METHOD PUBLIC CallBack : DINT
VAR_INPUT
  /// Response data
  RspData   : AxesGroupAcyclicAcrEntryRspBuffer;  
  /// Timestamp
  Timestamp : SystemTime;
END_VAR
// Create log entry
CreateLogMessage ( Timestamp   := Timestamp,
                   MessageType := MessageType.CMD,
                   Severity    := Severity.DEBUG,
                   MessageCode := 0,
                   MessageText := CONCAT('Callback reveiced in FB ', MyType));

ResponseData.Reset();
ResponseData.Payload    := RspData.Payload; 
ResponseData.PayloadLen := RspData.PayloadLen;
ParseResponsePayload( ResponseData :=  ResponseData , Timestamp := Timestamp);

// set flag for response received
_responseReceived := TRUE;
END_METHOD

METHOD PROTECTED CheckFunctionSupported : BOOL
VAR_IN_OUT
  /// Robot assignment of function
  AxesGroup : AxesGroup; 
END_VAR
Error   := TRUE;
ErrorID := RobotLibraryEvents.ERR_FUNCTION_NOT_SUPPORTED;

// Create log entry
CreateLogMessagePara1 ( Timestamp   := AxesGroup.InternalData.SystemTime,
                        MessageType := MessageType.CMD,
                        Severity    := Severity.DEBUG,
                        MessageCode := 0,
                        MessageText := 'Execution canceled, because function <{1}> is not supported by the robot controller',
                        Para1       :=  _myType);
END_METHOD

METHOD PROTECTED CheckParameterChanged : BOOL
VAR_IN_OUT
  /// Robot assignment of function
  AxesGroup    : AxesGroup; 
END_VAR
IF ( CheckParameterChanged )
THEN
  AxesGroup.Acyclic.ActiveCommandRegister.NotifyParameterChanged := _uniqueID;
END_IF
END_METHOD

METHOD PROTECTED CheckParameterValid : BOOL
VAR_IN_OUT
  /// Robot assignment of function
  AxesGroup : AxesGroup; 
END_VAR
CheckParameterValid := TRUE;
END_METHOD

METHOD INTERNAL CreateCommandPayload : RobotLibrarySendDataFB
VAR_IN_OUT
  /// Robot assignment of function
  AxesGroup    : AxesGroup; 
END_VAR
// Reset all variables
CreateCommandPayload.Reset();
// Add CmdType
CreateCommandPayload.AddUint(_cmdHeader.CmdTyp);
// Add Reserve_ExecMode
CreateCommandPayload.AddHalfBytes(  0               , _cmdHeader.ExecMode);
// Add ParSeq_Priority
CreateCommandPayload.AddHalfBytes( _cmdHeader.ParSeq, _cmdHeader.Priority);
END_METHOD

METHOD PROTECTED OnCall
VAR_IN_OUT
  /// Robot assignment of function
  AxesGroup         : AxesGroup; 
END_VAR
// map numeric value to enum, so that the corresponding message text is directly shown by the tooltip
ErrorIdEnum   := ErrorId;
WarningIdEnum := WarningId;
InfoIdEnum    := InfoId;

Error := ErrorID <> RobotLibraryConstants.OK;

ExternalLogger := AxesGroup.MessageLog.ExternalLogger;
LogLevel       := AxesGroup.MessageLog.LogLevel;

// building rising edges for error, warning, info number detected
_error_R  ( CLK := ErrorID   <> RobotLibraryConstants.OK );
_warning_R( CLK := WarningID <> RobotLibraryConstants.OK );
_info_R   ( CLK := InfoID    <> RobotLibraryConstants.OK );

IF ( _error_R.Q)
THEN
  // Create log entry
  CreateLogMessagePara2 ( Timestamp   := AxesGroup.InternalData.SystemTime,
                          MessageType := MessageType.CMD,
                          Severity    := Severity.DEBUG,
                          MessageCode := 0,
                          MessageText := 'Error with ID: 16#{1} in FB {2} received ',
                          Para1       := WORD_TO_STRING_HEX(ErrorID),
                          Para2       := MyType);                        
END_IF

IF ( _warning_R.Q)
THEN
  // Create log entry
  CreateLogMessagePara2 ( Timestamp   := AxesGroup.InternalData.SystemTime,
                          MessageType := MessageType.CMD,
                          Severity    := Severity.DEBUG,
                          MessageCode := 0,
                          MessageText := 'Warning with ID: 16#{1} in FB {2} received ',
                          Para1       := WORD_TO_STRING_HEX(WarningID),
                          Para2       := MyType);                        
END_IF

IF ( _info_R.Q)
THEN
  // Create log entry
  CreateLogMessagePara2 ( Timestamp   := AxesGroup.InternalData.SystemTime,
                          MessageType := MessageType.CMD,
                          Severity    := Severity.DEBUG,
                          MessageCode := 0,
                          MessageText := 'Info with ID: 16#{1} in FB {2} received ',
                          Para1       := WORD_TO_STRING_HEX(InfoID),
                          Para2       := MyType);                        
END_IF
END_METHOD

METHOD OnOnlineChange : DINT
VAR_IN_OUT
  /// Robot assignment of function
  AxesGroup : AxesGroup; 
END_VAR
// update pointer to command FB
AxesGroup.Acyclic.ActiveCommandRegister.OnOnlineChange( UniqueID := _uniqueID, pCommandFB := ADR(THIS^));
END_METHOD

METHOD INTERNAL ParseResponsePayload : DINT
VAR_INPUT
  /// Response data
  ResponseData : RobotLibraryRecvDataFB;
  /// Timestamp
  Timestamp    : SystemTime;  
END_VAR
// reset message IDs 
InfoID    := 0;
WarningID := 0;
ErrorID   := 0;

// get State
_rspHeader.State                := ResponseData.GetHalfeByte1(IncPayloadPtr := FALSE);
// get ParSeq
_rspHeader.ParSeq               := ResponseData.GetHalfeByte2(IncPayloadPtr := TRUE);
// get AlarmMessageSeverity
_rspHeader.AlarmMessageSeverity := ResponseData.GetSint();
// get AlarmMessageCode
_rspHeader.AlarmMessageCode     := ResponseData.GetUint();


// Update InfoID / WarningID / ErrorID
CASE _rspHeader.AlarmMessageSeverity OF

  // Informative message
  Severity.INFO        : InfoID    := _rspHeader.AlarmMessageCode;
  // Warning message
  Severity.WARNING     : WarningID := _rspHeader.AlarmMessageCode;
  // Error message
  Severity.ERROR       : ErrorID   := _rspHeader.AlarmMessageCode; 
  // Fataö error message
  Severity.FATAL_ERROR : ErrorID   := _rspHeader.AlarmMessageCode;

END_CASE

ParseResponsePayload := ResponseData.PayloadPtr;
END_METHOD

METHOD PROTECTED Reset : DINT
VAR_INPUT
END_VAR
_parameterUpdateInternal := FALSE;
_uniqueId := 0;
_stepCmd  := 0;
Error     := FALSE;
ErrorID   := 0;
WarningID := 0;
InfoID    := 0;  

Reset := RobotLibraryConstants.OK;
END_METHOD

END_FUNCTION_BLOCK

// Library/POUs/_internal/RobotLibraryRecvDataFB
{attribute 'pack_mode' := '1'} 
FUNCTION_BLOCK RobotLibraryRecvDataFB
// ------------------------------------------------------------------------- 
//  SRCI Robot Library                                                
// ------------------------------------------------------------------------- 
//                                                                           
//  Object:      RecvData                                       
//  Author:      Thorsten Brach                                                
//  Date:        2024-06-01
//
//  Description:                                              
//   
//                                                                           
//  Copyright: 
//    (C) 2024 Thorsten Brach. All rights reserved                                                                                                                                            
//             Licensed under the LGPL-3.0 license.
//                                                                           
//  Disclaimer:                                                                           
//    This project is provided without any guarantee and can be used for   
//    private and commercial purposes. Any use is at the user’s 
//    own risk and responsibility.
//
// -------------------------------------------------------------------------
VAR_INPUT
  /// Payload
  Payload    : ARRAY [0..RobotLibraryParameter.TELEGRAM_PAYLOAD_MAX] OF BYTE;
  /// Payload length
  PayloadLen : UDINT;
  /// Payload pointer
  PayloadPtr : DINT;
END_VAR

/// returns a ArmConfigParameter from the payload buffer from the current payload pointer address and increase the payload pointer afterwards
METHOD GetArmConfig : ArmConfigParameter
VAR
  /// temporary byte
 _tmpByte : BYTE;
END_VAR
// Table 5-17: Meaning of “Config” byte
// BIT 0 Shoulder TRUE : Shoulder is Back
//                FALSE: Shoulder is Front
// BIT 1 Elbow    TRUE : Elbow is Down
//                FALSE: Elbow is Up
// BIT 2 Wrist    TRUE : Wrist is Flip
//                FALSE: Wrist is Non-Flip
// BIT 3 Spare Not used
// BIT 4 Spare Not Used
// BIT 5 Spare Not Used
// BIT 6 Spare Not Used
// BIT 7 Spare Not Used
// get 1st Byte
_tmpByte := GetByte();

IF ( _tmpByte.0 ) 
THEN
  GetArmConfig.Shoulder := ArmConfigShoulder.BACK;
ELSE
  GetArmConfig.Shoulder := ArmConfigShoulder.FRONT;
END_IF

IF ( _tmpByte.1 ) 
THEN
  GetArmConfig.Elbow := ArmConfigElbow.DOWN;
ELSE
  GetArmConfig.Elbow := ArmConfigElbow.UP;
END_IF

IF ( _tmpByte.2 ) 
THEN
  GetArmConfig.Wrist := ArmConfigWrist.FLIP;
ELSE
  GetArmConfig.Wrist := ArmConfigWrist.NON_FLIP;
END_IF


// get 2nd byte to inc the PayloadPointer
_tmpByte := GetByte();
END_METHOD

/// returns a BOOL from the payload buffer from the current payload pointer address and increase the payload pointer afterwards
METHOD GetBool : BOOL
// copy data
GetBool := Payload[PayloadPtr].0;
// inc payload pointer 
PayloadPtr := PayloadPtr + SIZEOF(BYTE);
END_METHOD

/// returns a BYTE from the payload buffer from the current payload pointer address and increase the payload pointer afterwards
METHOD GetByte : BYTE
// copy data
GetByte := Payload[PayloadPtr];
// inc payload pointer 
PayloadPtr := PayloadPtr + SIZEOF(BYTE);
END_METHOD

/// returns a datablock from the payload buffer from the current payload pointer address and increase the payload pointer afterwards
METHOD GetDataBlock
VAR_INPUT
  /// Target
  pData    : POINTER TO BYTE;
  /// Size of data block
  Size     : UDINT;
  /// Target data type is string ? 
  IsString : BOOL;
END_VAR
IF ( pData <> RobotLibraryConstants.NULL_POINTER)
THEN
  IF ( IsString)
  THEN
    Size := Size -1;
  END_IF

  // copy data
  SysDepMemCpy(pDest := pData, pSrc := ADR(Payload[PayloadPtr]), DataLen := Size);
  
  // inc payload pointer 
  PayloadPtr := PayloadPtr + UDINT_TO_DINT(Size);
END_IF
END_METHOD

/// returns a DataInSync from the payload buffer from the current payload pointer address and increase the payload pointer afterwards
METHOD GetDataInSync : DataInSync
VAR
  /// temporary byte
 _tmpByte : BYTE;
END_VAR
// copy data
_tmpByte := Payload[PayloadPtr];

GetDataInSync.ToolsInSync             := _tmpByte.0;
GetDataInSync.FramesInSync            := _tmpByte.1;
GetDataInSync.LoadsInSync             := _tmpByte.2;
GetDataInSync.WorkAreasInSync         := _tmpByte.3;
GetDataInSync.SoftwareLimitsInSync    := _tmpByte.4;
GetDataInSync.DefaultDynamicsInSync   := _tmpByte.5;
GetDataInSync.ReferenceDynamicsInSync := _tmpByte.6;

// inc payload pointer   
PayloadPtr := PayloadPtr + SIZEOF(BYTE);
END_METHOD

/// returns a DWORD from the payload buffer from the current payload pointer address and increase the payload pointer afterwards
METHOD GetDword : DWORD
// copy data
SysDepMemCpy(pDest := ADR(GetDword), pSrc := ADR(Payload[PayloadPtr]), DataLen := SIZEOF(DWORD));
// inc payload pointer 
PayloadPtr := PayloadPtr + SIZEOF(DWORD);
END_METHOD

/// returns a FragmentAction from the payload buffer from the current payload pointer address and increase the payload pointer afterwards
METHOD GetFragmentAction : FragmentAction
VAR
  /// temporary byte
 _tmpByte : BYTE;
END_VAR
// copy data
_tmpByte := Payload[PayloadPtr];

GetFragmentAction.Complete := _tmpByte.0;
GetFragmentAction.Reset    := _tmpByte.1;
GetFragmentAction.Clear    := _tmpByte.2;
GetFragmentAction.BIT03    := _tmpByte.3;
GetFragmentAction.BIT04    := _tmpByte.4;
GetFragmentAction.BIT05    := _tmpByte.5;
GetFragmentAction.BIT06    := _tmpByte.6;
GetFragmentAction.BIT07    := _tmpByte.7;

// inc payload pointer   
PayloadPtr := PayloadPtr + SIZEOF(BYTE);
END_METHOD

/// returns the 1st halfe BYTE from the payload buffer from the current payload pointer address and increase the payload pointer afterwards
METHOD GetHalfeByte1 : BYTE
VAR_INPUT
  /// Increase payload pointer 
  IncPayloadPtr : BOOL;
END_VAR

VAR
  /// temporary byte
 _tmpByte : BYTE;
END_VAR
// copy data
_tmpByte := Payload[PayloadPtr];

GetHalfeByte1.0 := _tmpByte.0;
GetHalfeByte1.1 := _tmpByte.1;
GetHalfeByte1.2 := _tmpByte.2;
GetHalfeByte1.3 := _tmpByte.3;


IF (IncPayloadPtr)
THEN  
  // inc payload pointer
  PayloadPtr := PayloadPtr + SIZEOF(BYTE);
END_IF
END_METHOD

/// returns the 1st halfe BYTE from the payload buffer from the current payload pointer address and increase the payload pointer afterwards
METHOD GetHalfeByte2 : BYTE
VAR_INPUT
  /// Increase payload pointer 
  IncPayloadPtr : BOOL;
END_VAR

VAR
  /// temporary byte
 _tmpByte : BYTE;
END_VAR
// copy data
_tmpByte := Payload[PayloadPtr];

GetHalfeByte2.0 := _tmpByte.4;
GetHalfeByte2.1 := _tmpByte.5;
GetHalfeByte2.2 := _tmpByte.6;
GetHalfeByte2.3 := _tmpByte.7;

IF (IncPayloadPtr)
THEN  
  // inc payload pointer
  PayloadPtr := PayloadPtr + SIZEOF(BYTE);
END_IF
END_METHOD

/// returns a IEC_Date from the payload buffer from the current payload pointer address and increase the payload pointer afterwards
METHOD GetIecDate : IEC_Date
// copy data
SysDepMemCpy(pDest := ADR(GetIecDate), pSrc := ADR(Payload[PayloadPtr]), DataLen := SIZEOF(IEC_DATE));
// swap byte order
GetIecDate := SwapIecDate(GetIecDate);
// inc payload pointer   
PayloadPtr := PayloadPtr + SIZEOF(IEC_DATE);
END_METHOD

/// returns a IEC_TIME from the payload buffer from the current payload pointer address and increase the payload pointer afterwards
METHOD GetIecTime : IEC_TIME
// copy data
SysDepMemCpy(pDest := ADR(GetIecTime), pSrc := ADR(Payload[PayloadPtr]), DataLen := SIZEOF(IEC_TIME));
// swap byte order
GetIecTime := SwapIecTime(GetIecTime);
// inc payload pointer   
PayloadPtr := PayloadPtr + SIZEOF(IEC_TIME);
END_METHOD

/// returns a INT from the payload buffer from the current payload pointer address and increase the payload pointer afterwards
METHOD GetInt : INT
// copy data
SysDepMemCpy(pDest := ADR(GetInt), pSrc := ADR(Payload[PayloadPtr]), DataLen := SIZEOF(INT));
// swap byte order
GetInt := SwapInt(GetInt);
// inc payload pointer   
PayloadPtr := PayloadPtr + SIZEOF(INT);
END_METHOD

/// returns a REAL from the payload buffer from the current payload pointer address and increase the payload pointer afterwards
METHOD GetReal : REAL
// copy data
SysDepMemCpy(pDest := ADR(GetReal), pSrc := ADR(Payload[PayloadPtr]), DataLen := SIZEOF(REAL));
// swap byte order
GetReal := SwapReal(GetReal);
// inc payload pointer   
PayloadPtr := PayloadPtr + SIZEOF(Real);
END_METHOD

/// returns a SINT from the payload buffer from the current payload pointer address and increase the payload pointer afterwards
METHOD GetSint : SINT
// copy data
SysDepMemCpy(pDest := ADR(GetSint), pSrc := ADR(Payload[PayloadPtr]), DataLen := SIZEOF(SINT));
// inc payload pointer 
PayloadPtr := PayloadPtr + SIZEOF(SINT);
END_METHOD

/// returns a String from the payload buffer from the current payload pointer address and increase the payload pointer afterwards
METHOD GetString : STRING(255)
VAR_INPUT
  Size : DINT;
END_VAR
// copy data
SysDepMemCpy(pDest := ADR(GetString), pSrc := ADR(Payload[PayloadPtr]), DataLen := DINT_TO_UDINT(Size));

// inc payload pointer 
PayloadPtr := PayloadPtr + Size;
END_METHOD

/// returns a TrackingStatus from the payload buffer from the current payload pointer address and increase the payload pointer afterwards
METHOD GetTrackingStatus : TrackingStatus
VAR
  /// temporary byte
  tmpByte : BYTE;
END_VAR
// copy data
tmpByte := GetByte();

GetTrackingStatus.ConveyorTrackingEnabled   := tmpByte.0;  
GetTrackingStatus.WaitingForSynchronization := tmpByte.1;
GetTrackingStatus.Synchronizing             := tmpByte.2;
GetTrackingStatus.Synchronous               := tmpByte.3;
GetTrackingStatus.Desynchronizing           := tmpByte.4;
GetTrackingStatus.SyncOutZoneEntered        := tmpByte.5;
GetTrackingStatus.SyncOutZoneLeft           := tmpByte.6;
GetTrackingStatus.NotUsed                   := tmpByte.7;
END_METHOD

/// returns a TurnNumber from the payload buffer from the current payload pointer address and increase the payload pointer afterwards
METHOD GetTurnNumbers : TurnNumber
GetTurnNumbers.J1Turns := BYTE_TO_SINT(GetHalfeByte1(FALSE));
GetTurnNumbers.J2Turns := BYTE_TO_SINT(GetHalfeByte2(TRUE));

GetTurnNumbers.J3Turns := BYTE_TO_SINT(GetHalfeByte1(FALSE));
GetTurnNumbers.J4Turns := BYTE_TO_SINT(GetHalfeByte2(TRUE));

GetTurnNumbers.J5Turns := BYTE_TO_SINT(GetHalfeByte1(FALSE));
GetTurnNumbers.J6Turns := BYTE_TO_SINT(GetHalfeByte2(TRUE));

GetTurnNumbers.E1Turns := BYTE_TO_SINT(GetByte());
END_METHOD

/// returns a UDINT from the payload buffer from the current payload pointer address and increase the payload pointer afterwards
METHOD GetUdint : UDINT
// copy data
SysDepMemCpy(pDest := ADR(GetUdint), pSrc := ADR(Payload[PayloadPtr]), DataLen := SIZEOF(UDINT));
// swap byte order
GetUdint := SwapUdint(GetUdint);
// inc payload pointer   
PayloadPtr := PayloadPtr + SIZEOF(UDINT);
END_METHOD

/// returns a UINT from the payload buffer from the current payload pointer address and increase the payload pointer afterwards
METHOD GetUint : UINT
// copy data
SysDepMemCpy(pDest := ADR(GetUint), pSrc := ADR(Payload[PayloadPtr]), DataLen := SIZEOF(UINT));
// swap byte order
GetUint := SwapUint(GetUint);
// inc payload pointer   
PayloadPtr := PayloadPtr + SIZEOF(UINT);
END_METHOD

/// returns a USINT from the payload buffer from the current payload pointer address and increase the payload pointer afterwards
METHOD GetUsint : USINT
// copy data
SysDepMemCpy(pDest := ADR(GetUsint), pSrc := ADR(Payload[PayloadPtr]), DataLen := SIZEOF(USINT));
// inc payload pointer 
PayloadPtr := PayloadPtr + SIZEOF(USINT);
END_METHOD

/// returns a WORD from the payload buffer from the current payload pointer address and increase the payload pointer afterwards
METHOD GetWord : WORD
// copy data
SysDepMemCpy(pDest := ADR(GetWord), pSrc := ADR(Payload[PayloadPtr]), DataLen := SIZEOF(WORD));
// swap byte order
GetWord := SwapWord(GetWord);
// inc payload pointer   
PayloadPtr := PayloadPtr + SIZEOF(WORD);
END_METHOD

/// Resets the payload buffer, the payload pointer and the payload length
METHOD Reset
VAR_INPUT
END_VAR
SysDepMemSet(pDest := ADR(Payload), Value := 0 , DataLen := SIZEOF(Payload));
PayloadLen := 0;
PayloadPtr := 0;
END_METHOD

END_FUNCTION_BLOCK

// Library/POUs/_internal/AxesGroupMessageLogFB
FUNCTION_BLOCK AxesGroupMessageLogFB
// ------------------------------------------------------------------------- 
//  SRCI Robot Library                                                
// ------------------------------------------------------------------------- 
//                                                                           
//  Object:      AxesGroupMessageLogFB                                       
//  Author:      Thorsten Brach                                                
//  Date:        2025-01-05
//
//  Description:                                              
//   
//                                                                           
//  Copyright: 
//    (C) 2025 Thorsten Brach. All rights reserved                                                                                                                                            
//             Licensed under the LGPL-3.0 license.
//                                                                           
//  Disclaimer:                                                                           
//    This project is provided without any guarantee and can be used for   
//    private and commercial purposes. Any use is at the user’s 
//    own risk and responsibility.
//
// -------------------------------------------------------------------------
VAR_INPUT
  /// Logging level
  LogLevel         : LogLevel;
  /// Interface to an external logger
  ExternalLogger   : IMessageLogger;
END_VAR


VAR_OUTPUT
  /// Amount of system log entries
  SystemLogEntries : UINT := 0;
  /// Amount of message log entries
  MessagesEntries  : UINT := 0;
  /// System log
  SystemLogs       : ARRAY[0..RobotLibraryParameter.SYSTEM_LOG_MAX] OF STRING(255);
  /// Message Log
  Messages         : ARRAY[0..RobotLibraryParameter.MESSAGE_LOG_MAX] OF AlarmMessage;  
END_VAR

METHOD PUBLIC AddMessage
VAR_INPUT
  Message : ReadMessagesRecvData;
END_VAR

VAR
  /// internal index
 _idx            : DINT;
  /// internal index to delete
 _idxFound       : DINT;
  /// lowest Severity
 _lowestSeverity : Severity := Severity.FATAL_ERROR;
END_VAR
// Check entry must be added ? 
IF (( LogLevel  <= Message.Severity        ) AND
    ( LogLevel  >  LogLevelEnum.DEACTIVATE ))
THEN
  // Check message buffer is full ? 
  IF ( MessagesEntries >= RobotLibraryParameter.MESSAGE_LOG_MAX )
  THEN
    // find lowest Severity
    FOR _idx := 1 TO RobotLibraryParameter.MESSAGE_LOG_MAX
    DO
      // check entry has a lower severity ? 
     _lowestSeverity := MIN( Messages[_idx].Severity, _lowestSeverity );
		END_FOR

    // search for the oldes message with a lower Severity 
    FOR _idx := RobotLibraryParameter.MESSAGE_LOG_MAX TO 1 BY -1
    DO
      // message found ?
      IF (( Messages[_idx].Severity <  Message.Severity ) AND
          ( Messages[_idx].Severity <=  _lowestSeverity ))
      THEN
        // save index to delete 
       _idxFound := _idx;
        EXIT;
			END_IF
		END_FOR
    
    // check message must be deleted ? 
    IF ( _idxFound > 0 )
    THEN
      // shift all messages starting from the found index one position forwards
      FOR _idx := _idxFound TO RobotLibraryParameter.MESSAGE_LOG_MAX -1
      DO
        Messages[_idx] := Messages[_idx +1];
			END_FOR
		END_IF
  END_IF  


  // shift all messages one position backwards
  FOR _idx := RobotLibraryParameter.MESSAGE_LOG_MAX TO 1 BY -1
  DO
    Messages[_idx] := Messages[_idx-1]; 
  END_FOR

  // Add new message 
  Messages[0].Timestamp.SystemDate := IEC_DATE_TO_DATE(Message.Timestamp.IEC_DATE);           
  Messages[0].Timestamp.SystemTime := IEC_TIME_TO_TIME(Message.Timestamp.IEC_TIME);           
  Messages[0].MessageType          :=                  Message.MsgType;
  Messages[0].Severity             :=                  Message.Severity;
  Messages[0].MessageText          :=                  Message.Text;
  Messages[0].MessageCode          :=                  Message.ErrorCode;
  
  // inc message counter
  MessagesEntries := DINT_TO_UINT(LIMIT(0, MessagesEntries + 1, RobotLibraryParameter.MESSAGE_LOG_MAX));
END_IF
END_METHOD

METHOD PUBLIC AddSystemLog
VAR_INPUT
  SystemLog : STRING(255);
END_VAR

VAR
  /// internal index
 _idx : DINT;
END_VAR
FOR _idx := RobotLibraryParameter.SYSTEM_LOG_MAX TO 1 BY -1
DO
  SystemLogs[_idx] := SystemLogs[_idx-1]; 
END_FOR

SystemLogs[0] := SystemLog;           

// inc SystemLog counter
SystemLogEntries := DINT_TO_UINT(LIMIT(0, SystemLogEntries + 1, RobotLibraryParameter.SYSTEM_LOG_MAX));
END_METHOD

METHOD PUBLIC DeleteMessages
VAR_INPUT
END_VAR
// reset messages
SysDepMemSet(ADR(Messages), 0, SIZEOF(Messages));
// reset message counter
MessagesEntries := 0;
END_METHOD

METHOD DeleteSystemLogs
VAR_INPUT
END_VAR
// reset SystemLogs
SysDepMemSet(ADR(SystemLogs), 0, SIZEOF(SystemLogs));
// reset SystemLogs counter
SystemLogEntries := 0;
END_METHOD

END_FUNCTION_BLOCK

// Library/POUs/_internal/RobotLibraryBaseEnableFB
FUNCTION_BLOCK RobotLibraryBaseEnableFB EXTENDS RobotLibraryBaseFB
// ------------------------------------------------------------------------- 
//  SRCI Robot Library                                                
// ------------------------------------------------------------------------- 
//                                                                           
//  Object:      RobotLibraryBaseFB                                       
//  Author:      Thorsten Brach                                                
//  Date:        2024-08-11
//
//  Description:                                              
//   
//                                                                           
//  Copyright: 
//    (C) 2024 Thorsten Brach. All rights reserved                                                                                                                                            
//             Licensed under the LGPL-3.0 license.
//                                                                           
//  Disclaimer:                                                                           
//    This project is provided without any guarantee and can be used for   
//    private and commercial purposes. Any use is at the user’s 
//    own risk and responsibility.
//
// -------------------------------------------------------------------------
VAR_INPUT
  /// Set TRUE to activate / Set False to deactivate
  Enable            : BOOL;
END_VAR

VAR_OUTPUT
  /// FB is being processed
  Busy              : BOOL;
  /// Command is transferred and confirmed by the RC
//CommandBuffered   : BOOL;
  /// TRUE while function is active
  Enabled           : BOOL;
  /// Receiving of input parameter values has been acknowledged by RC
//ParameterAccepted : BOOL;
END_VAR

VAR
  /// step counter for finite state machine
 _fsmState          : FsmState;
  /// Rising edge for enable
 _enable_R          : R_TRIG;
  /// Falling edge for enable
 _enable_F          : F_TRIG;
END_VAR

SUPER^(AxesGroup := AxesGroup);

METHOD INTERNAL FSM : DINT
VAR_IN_OUT
  /// Robot assignment of function
  AxesGroup : AxesGroup; 
END_VAR
VAR
  /// internal return value
 _retVal : DINT;
END_VAR
CASE _fsmState 
OF

  FsmState.READY :
  
    // Await start
    IF (( NOT Busy       ) AND 
        ( NOT Error      ) AND 
        (    _enable_R.Q ))
    THEN
      // inc fsm step
     _fsmState := FsmState.START;
    END_IF
      
  FsmState.START :
   
   _retVal := OnExecStart(AxesGroup := AxesGroup);
    
    IF ( _retVal = RobotLibraryConstants.OK )
    THEN
     _fsmState := FsmState.RUNNING;
    ELSE
      // Cancel
      IF ((      Busy       ) AND
          (  NOT Error      ) AND
          (     _enable_F.Q ))
      THEN
       _fsmState := FsmState.CANCEL;
        RETURN;
      END_IF
    
      // check error 
      IF (_retVal < RobotLibraryConstants.OK)
      THEN
       _fsmState := FsmState.ERROR;
        RETURN;
      END_IF
    END_IF

   FsmState.RUNNING :

      _retVal := OnExecRun(AxesGroup := AxesGroup);
    
       IF (_retVal = RobotLibraryConstants.OK )
       THEN
        _fsmState := FsmState.DONE;
       ELSE
         // Cancel
         IF ((      Busy       ) AND
             (  NOT Error      ) AND
             (     _enable_F.Q ))
         THEN
          _fsmState := FsmState.CANCEL;
           RETURN;
         END_IF
         
         // error 
         IF (_retVal < RobotLibraryConstants.OK)
         THEN
          _fsmState := 99;
           RETURN;
         END_IF         
       END_IF

  FsmState.DONE :
  
   _fsmState := FsmState.READY;

  FsmState.CANCEL :

   _retVal := OnExecCancel(AxesGroup := AxesGroup);
    
    IF (_retVal = RobotLibraryConstants.OK )
    THEN
      _fsmState := FsmState.READY;
    END_IF
    
  FsmState.ERROR :
  
    IF (NOT Enable)
    THEN
     _fsmState := FsmState.ERROR_CLEAR;
    END_IF

  FsmState.ERROR_CLEAR :

   _retVal := OnExecErrorClear(AxesGroup := AxesGroup);
    
    IF (_retVal = RobotLibraryConstants.OK )
    THEN
      _fsmState := FsmState.READY;
    END_IF
       
ELSE
  ;
END_CASE
END_METHOD

METHOD PROTECTED OnCall
VAR_IN_OUT
  /// Robot assignment of function
  AxesGroup         : AxesGroup; 
END_VAR
SUPER^.OnCall(AxesGroup := AxesGroup);

// building rising and falling edges
_enable_R( CLK := Enable);
_enable_F( CLK := Enable);

// call state machine
FSM(AxesGroup := AxesGroup);


// Abort execution 
IF (Busy) AND ( _enable_F.Q) 
THEN
  // try to remove cmd
  AxesGroup.Acyclic.ActiveCommandRegister.RemoveCmd(_uniqueID);
END_IF
END_METHOD

METHOD Protected OnExecCancel : DINT
VAR_IN_OUT
  /// Robot assignment of function
  AxesGroup : AxesGroup; 
END_VAR
OnExecCancel := Reset();


// Create log entry
CreateLogMessagePara1 ( Timestamp   := AxesGroup.InternalData.SystemTime,
                        MessageType := MessageType.CMD,
                        Severity    := Severity.DEBUG,
                        MessageCode := 0,
                        MessageText := 'Execution of FB {1} cancled ',
                        Para1       := MyType);
END_METHOD

METHOD PROTECTED OnExecErrorClear : DINT
VAR_IN_OUT
  /// Robot assignment of function
  AxesGroup : AxesGroup; 
END_VAR
Reset();
END_METHOD

METHOD PROTECTED OnExecRun : DINT
VAR_IN_OUT
  /// Robot assignment of function
  AxesGroup : AxesGroup; 
END_VAR
END_METHOD

METHOD PROTECTED OnExecStart : DINT
VAR_IN_OUT
  /// Robot assignment of function
  AxesGroup : AxesGroup; 
END_VAR
END_METHOD

METHOD PROTECTED Reset : DINT
VAR_INPUT
END_VAR
Reset := SUPER^.Reset();

Busy    := FALSE;
Enabled := FALSE;
END_METHOD

END_FUNCTION_BLOCK

// Library/POUs/_internal/RobotLibraryBaseExecuteFB
FUNCTION_BLOCK RobotLibraryBaseExecuteFB EXTENDS RobotLibraryBaseFB
// ------------------------------------------------------------------------- 
//  SRCI Robot Library                                                
// ------------------------------------------------------------------------- 
//                                                                           
//  Object:      RobotLibraryBaseFB                                       
//  Author:      Thorsten Brach                                                
//  Date:        2024-08-11
//
//  Description:                                              
//   
//                                                                           
//  Copyright: 
//    (C) 2024 Thorsten Brach. All rights reserved                                                                                                                                            
//             Licensed under the LGPL-3.0 license.
//                                                                           
//  Disclaimer:                                                                           
//    This project is provided without any guarantee and can be used for   
//    private and commercial purposes. Any use is at the user’s 
//    own risk and responsibility.
//
// -------------------------------------------------------------------------
VAR_INPUT
  /// Start of the command at the rising edge
  Execute         : BOOL;
END_VAR
VAR_OUTPUT
  /// The command has been completed successfully
  Done            : BOOL;
  /// FB is being processed
  Busy            : BOOL;
  /// Command is transferred and confirmed by the RC
//  CommandBuffered : BOOL;  
END_VAR


VAR
  /// step counter for finite state machine
 _fsmState        : FsmState;
  /// Rising edge for execute
 _execute_R       : R_TRIG;
  /// Falling edge for execute
 _execute_F       : F_TRIG;
END_VAR

SUPER^(AxesGroup := AxesGroup);

METHOD internal FSM : DINT
VAR_IN_OUT
  /// Robot assignment of function
  AxesGroup : AxesGroup; 
END_VAR
VAR
  /// internal return value
 _retVal : DINT;
END_VAR
CASE _fsmState 
OF

  FsmState.READY :
  
    // Await start
    IF (( NOT Busy        ) AND 
        ( NOT Error       ) AND 
        (    _execute_R.Q ))
    THEN
      // inc fsm step
     _fsmState := FsmState.START;
    END_IF
      
  FsmState.START :
   
   _retVal := OnExecStart(AxesGroup := AxesGroup);
    
    IF ( _retVal = RobotLibraryConstants.OK )
    THEN
     _fsmState := FsmState.RUNNING;
    ELSE
      // Cancel
      IF ((      Busy        ) AND
          (  NOT Error       ) AND
          (     _execute_F.Q ))
      THEN
       _fsmState := FsmState.CANCEL;
        RETURN;
      END_IF
    
      // check error 
      IF (_retVal < RobotLibraryConstants.OK)
      THEN
       _fsmState := FsmState.ERROR;
        RETURN;
      END_IF
    END_IF

   FsmState.RUNNING :

      _retVal := OnExecRun(AxesGroup := AxesGroup);
    
       IF (_retVal = RobotLibraryConstants.OK )
       THEN
        _fsmState := FsmState.DONE;
       ELSE
         // Cancel
         IF ((      Busy        ) AND
             (  NOT Error       ) AND
             (     _execute_F.Q ))
         THEN
          _fsmState := FsmState.CANCEL;
           RETURN;
         END_IF
         
         // error 
         IF (_retVal < RobotLibraryConstants.OK)
         THEN
          _fsmState := 99;
           RETURN;
         END_IF         
       END_IF

  FsmState.DONE :
  
   _fsmState := FsmState.READY;

  FsmState.CANCEL :

   _retVal := OnExecCancel(AxesGroup := AxesGroup);
    
    IF (_retVal = RobotLibraryConstants.OK )
    THEN
      _fsmState := FsmState.READY;
    END_IF
    
  FsmState.ERROR :
  
    IF (NOT Execute)
    THEN
     _fsmState := FsmState.ERROR_CLEAR;
    END_IF

  FsmState.ERROR_CLEAR :

   _retVal := OnExecErrorClear(AxesGroup := AxesGroup);
    
    IF (_retVal = RobotLibraryConstants.OK )
    THEN
      _fsmState := FsmState.READY;
    END_IF
       
ELSE
  ;
END_CASE
END_METHOD

// Base implementation must be called ! 
METHOD PROTECTED OnCall
VAR_IN_OUT
  /// Robot assignment of function
  AxesGroup         : AxesGroup; 
END_VAR
SUPER^.OnCall(AxesGroup := AxesGroup);

// building rising and falling edges
_execute_R( CLK := Execute);
_execute_F( CLK := EXecute);

// call state machine
FSM(AxesGroup := AxesGroup);

// Abort execution 
IF (Busy) AND (_execute_F.Q) 
THEN
  // try to remove cmd
  AxesGroup.Acyclic.ActiveCommandRegister.RemoveCmd(_uniqueID);
END_IF
END_METHOD

METHOD PROTECTED OnExecCancel : DINT
VAR_IN_OUT
  /// Robot assignment of function
  AxesGroup : AxesGroup; 
END_VAR
OnExecCancel := Reset();


// Create log entry
CreateLogMessagePara1 ( Timestamp   := AxesGroup.InternalData.SystemTime,
                        MessageType := MessageType.CMD,
                        Severity    := Severity.DEBUG,
                        MessageCode := 0,
                        MessageText := 'Execution of FB {1} cancled ',
                        Para1       := MyType);
END_METHOD

METHOD PROTECTED OnExecErrorClear : DINT
VAR_IN_OUT
  /// Robot assignment of function
  AxesGroup : AxesGroup; 
END_VAR
Reset();
END_METHOD

METHOD PROTECTED OnExecRun : DINT
VAR_IN_OUT
  /// Robot assignment of function
  AxesGroup : AxesGroup; 
END_VAR
END_METHOD

METHOD PROTECTED OnExecStart : DINT
VAR_IN_OUT
  /// Robot assignment of function
  AxesGroup : AxesGroup; 
END_VAR
END_METHOD

METHOD PROTECTED Reset : DINT
VAR_INPUT
END_VAR
Reset := SUPER^.Reset();

Done := FALSE;
Busy := FALSE;
END_METHOD

END_FUNCTION_BLOCK

// Library/POUs/Additional/MC_AbortMeasuringInput/MC_AbortMeasuringInputFB
/// Abort triggering of Position, measuring input
FUNCTION_BLOCK MC_AbortMeasuringInputFB EXTENDS RobotLibraryBaseExecuteFB
// ------------------------------------------------------------------------- 
//  SRCI Robot Library                                                
// ------------------------------------------------------------------------- 
//                                                                           
//  Object:      AbortMeasuringInputFB                                       
//  Author:      Thorsten Brach                                                
//  Date:        2024-06-01
//
//  Description:                                              
//   
//                                                                           
//  Copyright: 
//    (C) 2024 Thorsten Brach. All rights reserved                                                                                                                                            
//             Licensed under the LGPL-3.0 license.
//                                                                           
//  Disclaimer:                                                                           
//    This project is provided without any guarantee and can be used for   
//    private and commercial purposes. Any use is at the user’s 
//    own risk and responsibility.
//
// -------------------------------------------------------------------------
VAR_INPUT
  /// Command parameter 
  ParCmd          : AbortMeasuringInputParCmd;      
END_VAR
VAR_OUTPUT
  /// Command is transferred and confirmed by the RC
  CommandBuffered : BOOL;  
  /// Command output 
  OutCmd          : AbortMeasuringInputOutCmd;          
END_VAR
VAR
  /// internal copy of command parameter 
 _parCmd          : AbortMeasuringInputParCmd;
  /// command data to send
 _command         : AbortMeasuringInputSendData;
  /// response data received
 _response        : AbortMeasuringInputRecvData;      
END_VAR

SUPER^(AxesGroup := AxesGroup);

METHOD PROTECTED CheckFunctionSupported : BOOL
VAR_IN_OUT
  /// Robot assignment of function
  AxesGroup : AxesGroup; 
END_VAR
CheckFunctionSupported := AxesGroup.InternalData.RCSupportedFunctions.AbortMeasuringInput;

IF ( NOT CheckFunctionSupported )
THEN
  // call base implementation for set error and create log entry
  SUPER^.CheckFunctionSupported(AxesGroup := AxesGroup);
END_IF
END_METHOD

METHOD PROTECTED CheckParameterChanged : BOOL
VAR_IN_OUT
  /// Robot assignment of function
  AxesGroup    : AxesGroup; 
END_VAR
// Check ParCmd Size is > 0, because MemCmp does not work correctly with size = 0
IF (SIZEOF(ParCmd) = 0) 
THEN 
  RETURN;
END_IF

// compare memory 
_parameterChanged := ( SysDepMemCmp(pData1 := ADR(ParCmd), pData2 := ADR(_parCmd), DataLen := SIZEOF(ParCmd)) <> RobotLibraryConstants.OK );

// check parameter valid ?
_parameterValid   := CheckParameterValid( AxesGroup := AxesGroup );

IF ((  _parameterChanged        )  AND 
    (  _parameterValid          )) OR
    (  _parameterUpdateInternal )  
THEN  
  // reset internal flag for send parameter update
 _parameterUpdateInternal := FALSE;
  // update internal copy of parameters 
 _parCmd := ParCmd;
  // inc parameter sequence
 _command.ParSeq := _command.ParSeq + 1;
  // update command data  
  CommandData := CreateCommandPayload(AxesGroup := AxesGroup); // ( Access via reference to rCommandFB in ACR )
  // notify active command register 
  AxesGroup.Acyclic.ActiveCommandRegister.NotifyParameterChanged := _uniqueID;
END_IF
END_METHOD

METHOD INTERNAL CreateCommandPayload : RobotLibrarySendDataFB
VAR_IN_OUT
  /// Robot assignment of function
  AxesGroup : AxesGroup; 
END_VAR
// Table 6-571: Sent CMD payload (PLC to RC) of "AbortMeasuringInput"
// --------------------------
// Header
// --------------------------
// Byte 000 : UINT  - Type HB     
// Byte 001 :       - Type LB    
// Byte 002 : USINT - Reserve | ExecutionMode
// Byte 003 : USINT - ParSeq  | Priority
// --------------------------
// Datablock
// --------------------------
// Byte 004 : UINT       - MeasuringID LW HB
// Byte 005 :            - MeasuringID LW LB
// set command parameter 
_command.CmdTyp      :=  CmdType.AbortMeasuringInput;
_command.ExecMode    :=  ExecMode;
_command.ParSeq      := _command.ParSeq;
_command.Priority    :=  Priority;
                     
_command.MeasuringID := parCmd.MeasuringID;

// copy command data to header
_cmdHeader := _command;
// call base implementation to copy header to payload buffer
CreateCommandPayload := SUPER^.CreateCommandPayload(AxesGroup := AxesGroup);

// add command.MeasuringID
CreateCommandPayload.AddUint(_command.MeasuringID);

// Create logging
CreateCommandPayloadLog(AxesGroup := AxesGroup);
END_METHOD

METHOD INTERNAL CreateCommandPayloadLog
VAR_IN_OUT
  /// Robot assignment of function
  AxesGroup : AxesGroup; 
END_VAR
// Create log entry for Parameter start
CreateLogMessage      ( Timestamp   := AxesGroup.InternalData.SystemTime,
                        MessageType := MessageType.CMD,
                        Severity    := Severity.DEBUG,
                        MessageCode := 0,
                        MessageText := 'Create command payload with the following parameter(s) :');
  
// Create log entry for MeasuringID
CreateLogMessagePara1 ( Timestamp   := AxesGroup.InternalData.SystemTime,
                        MessageType := MessageType.CMD,
                        Severity    := Severity.DEBUG,
                        MessageCode := 0,
                        MessageText := 'Command.MeasuringID = {1}',
                        Para1       :=  UINT_TO_STRING(_command.MeasuringID));
END_METHOD

METHOD FB_init : BOOL
VAR_INPUT
  /// if TRUE, the retain variables are initialized (warm start / cold start)
  bInitRetains : BOOL; 
  /// if TRUE, the instance afterwards gets moved into the copy code (online change)
  bInCopyCode  : BOOL;  
END_VAR
MyType := 'MC_AbortMeasuringInputFB';

ExecMode := ExecutionMode.PARALLEL;
END_METHOD

METHOD PROTECTED OnCall
VAR_IN_OUT
  /// Robot assignment of function
  AxesGroup : AxesGroup; 
END_VAR
// call base implementation
SUPER^.OnCall(AxesGroup := AxesGroup);

CASE _stepCmd OF
  
  00:  IF ( _execute_R.Q ) 
       THEN
         // Check function is supported and parameter are valid ?
         IF (( CheckFunctionSupported( AxesGroup := AxesGroup )) AND
             ( CheckParameterValid   ( AxesGroup := AxesGroup )))      
         THEN
           // set busy flag
           Busy := TRUE;
           // Reset command outputs
           SysDepMemSet(pDest := ADR(OutCmd), Value := 0, DataLen := SIZEOF(OutCmd));         
           // apply command parameter
          _parCmd := ParCmd;
           // init parameter sequence
          _command.ParSeq := 1;
           // create command data
           CommandData := CreateCommandPayload(AxesGroup := AxesGroup);
           // Add command to active command register
          _uniqueID := AxesGroup.Acyclic.ActiveCommandRegister.AddCmd( pCommandFB := ADR(THIS^ ));     
           // set timeout
           SetTimeout(PT := _timeoutCmd, rTimer := _timerCmd);
           // inc step counter
          _stepCmd := _stepCmd + 1;
         END_IF 
       END_IF


  01:  // Wait for responce received
       IF ( _responseReceived )
       THEN
         // reset response received flag
        _responseReceived := FALSE;

         CASE  _response.State 
         OF
           CmdMessageState.BUFFERED    : CommandBuffered    := TRUE;
           CmdMessageState.DONE        : Done               := TRUE;
           CmdMessageState.ERROR       : Error              := TRUE;
         END_CASE
                
         // Done, Aborted or Error ?
         IF (_response.State >= CmdMessageState.DONE )
         THEN
           // Reset busy flag
           Busy := FALSE;
           // set timeout
           SetTimeout(PT := _timeoutCmd, rTimer := _timerCmd);
           // inc step counter
          _stepCmd := _stepCmd + 1; 
         END_IF
       END_IF


  02: IF ( NOT Execute)
      THEN
        Reset();
      END_IF     
ELSE
  // invalid step
  ErrorID := RobotLibraryEvents.ERR_INVALID_STEP;
END_CASE


// Reset FB
IF ( NOT Execute )
THEN
  Reset();
END_IF
END_METHOD

METHOD INTERNAL ParseResponsePayload : DINT
VAR_INPUT
  /// Response data
  ResponseData : RobotLibraryRecvDataFB;
  /// Timestamp
  Timestamp    : SystemTime;  
END_VAR
// Table 6-572: Received CMD payload (RC to PLC) of "AbortMeasuringInput"
// --------------------------
// Header
// --------------------------
// Byte 00 : USINT - ParSeq | State     
// Byte 01 : SINT  - AlarmMessageSeverity    
// Byte 02 : UINT  - AlarmMessageCode HB
// Byte 03 :       - AlarmMessageCode LB
// call base implementation to parse the header from payload buffer
ResponseData.PayloadPtr := SUPER^.ParseResponsePayload(ResponseData := ResponseData, Timestamp := Timestamp);

// copy parsed header to response
_response.ParSeq               := _rspHeader.ParSeq;
_response.State                := _rspHeader.State;
_response.AlarmMessageSeverity := _rspHeader.AlarmMessageSeverity;
_response.AlarmMessageCode     := _rspHeader.AlarmMessageCode;

// Create logging
ParseResponsePayloadLog(ResponseData := ResponseData, Timestamp := Timestamp);
END_METHOD

METHOD INTERNAL ParseResponsePayloadLog
VAR_INPUT
  /// Response data
  ResponseData : RobotLibraryRecvDataFB;
  /// Timestamp
  Timestamp    : SystemTime;  
END_VAR
// Create log entry for Parameter start
CreateLogMessage      ( Timestamp   := Timestamp,
                        MessageType := MessageType.CMD,
                        Severity    := Severity.DEBUG,
                        MessageCode := 0,
                        MessageText := 'Parsed the following parameter(s) from response data:');
                        
// Create log entry for no parameter 
CreateLogMessage      ( Timestamp   := Timestamp,
                        MessageType := MessageType.CMD,
                        Severity    := Severity.DEBUG,
                        MessageCode := 0,
                        MessageText := 'This command has no parameter to parse...');
END_METHOD

METHOD PROTECTED Reset : DINT
VAR_INPUT
END_VAR
Reset := SUPER^.Reset();

Done            := FALSE;
Busy            := FALSE;
CommandBuffered := FALSE;
END_METHOD

END_FUNCTION_BLOCK

// Library/POUs/Additional/MC_ActivateNextCommand/MC_ActivateNextCommandFB
/// Cancel currently active move command and continue with the next buffered command
FUNCTION_BLOCK MC_ActivateNextCommandFB EXTENDS RobotLibraryBaseExecuteFB
// ------------------------------------------------------------------------- 
//  SRCI Robot Library                                                
// ------------------------------------------------------------------------- 
//                                                                           
//  Object:      ActivateNextCommandFB                                       
//  Author:      Thorsten Brach                                                
//  Date:        2024-06-01
//
//  Description:                                              
//   
//                                                                           
//  Copyright: 
//    (C) 2024 Thorsten Brach. All rights reserved                                                                                                                                            
//             Licensed under the LGPL-3.0 license.
//                                                                           
//  Disclaimer:                                                                           
//    This project is provided without any guarantee and can be used for   
//    private and commercial purposes. Any use is at the user’s 
//    own risk and responsibility.
//
// -------------------------------------------------------------------------
VAR_INPUT
  /// Command parameter 
  ParCmd          : ActivateNextCommandParCmd;
END_VAR
VAR_OUTPUT
  /// Command is transferred and confirmed by the RC
  CommandBuffered : BOOL;
  /// command results
  OutCmd          : ActivateNextCommandOutCmd;
END_VAR

VAR
  /// internal copy of command parameter 
 _parCmd          : ActivateNextCommandParCmd;
  /// command data to send
 _command         : ActivateNextCommandSendData;
  /// response data received
 _response        : ActivateNextCommandRecvData;   
  /// Trigger related EmitterID
 _emitterID       : ARRAY[0..3] OF SINT;
END_VAR

SUPER^(AxesGroup := AxesGroup);

METHOD PROTECTED CheckFunctionSupported : BOOL
VAR_IN_OUT
  /// Robot assignment of function
  AxesGroup : AxesGroup; 
END_VAR
CheckFunctionSupported := AxesGroup.InternalData.RCSupportedFunctions.ActivateNextCommand;

IF ( NOT CheckFunctionSupported )
THEN
  // call base implementation for set error and create log entry
  SUPER^.CheckFunctionSupported(AxesGroup := AxesGroup);
END_IF
END_METHOD

METHOD PROTECTED CheckParameterChanged : BOOL
VAR_IN_OUT
  /// Robot assignment of function
  AxesGroup    : AxesGroup; 
END_VAR
// Check ParCmd Size is > 0, because MemCmp does not work correctly with size = 0
IF (SIZEOF(ParCmd) = 0) 
THEN 
  RETURN;
END_IF

// compare memory 
_parameterChanged := ( SysDepMemCmp(pData1 := ADR(ParCmd), pData2 := ADR(_parCmd), DataLen := SIZEOF(ParCmd)) <> RobotLibraryConstants.OK );

// check parameter valid ?
_parameterValid   := CheckParameterValid( AxesGroup := AxesGroup );

IF ((  _parameterChanged        )  AND 
    (  _parameterValid          )) OR
    (  _parameterUpdateInternal )  
THEN  
  // reset internal flag for send parameter update
 _parameterUpdateInternal := FALSE;
  // update internal copy of parameters 
 _parCmd := ParCmd;
  // inc parameter sequence
 _command.ParSeq := _command.ParSeq + 1;
  // update command data  
  CommandData := CreateCommandPayload(AxesGroup := AxesGroup); // ( Access via reference to rCommandFB in ACR )
  // notify active command register 
  AxesGroup.Acyclic.ActiveCommandRegister.NotifyParameterChanged := _uniqueID;  
END_IF
END_METHOD

METHOD INTERNAL CreateCommandPayload : RobotLibrarySendDataFB
VAR_IN_OUT
  /// Robot assignment of function
  AxesGroup : AxesGroup; 
END_VAR
// Table 6-662: Sent CMD payload (PLC to RC) of "ActivateNextCommand"
// --------------------------
// Header
// --------------------------
// Byte 00 : UINT  - Type HB     
// Byte 01 :       - Type LB    
// Byte 02 : USINT - Reserve | ExecutionMode
// Byte 03 : USINT - ParSeq  | Priority
// --------------------------
// Datablock
// --------------------------
// Byte 04 : SINT - EmitterID[0]
// Byte 05 : SINT - EmitterID[1]
// Byte 06 : SINT - EmitterID[2]   
// Byte 07 : SINT - EmitterID[3]
// Byte 08 : SINT - ListenerID
// Byte 09 : BYTE - Reserve
// --------------------------
// set command parameter 
_command.CmdTyp     :=  CmdType.ActivateNextCommand;
_command.ExecMode   :=  ExecMode;
_command.ParSeq     := _command.ParSeq;
_command.Priority   :=  Priority;
_command.ListenerID := _parCmd.ListenerID;


// copy command data to header
_cmdHeader := _command;
// call base implementation to copy header to payload buffer
CreateCommandPayload := SUPER^.CreateCommandPayload(AxesGroup := AxesGroup);

// add command.EmitterID[0]
CreateCommandPayload.AddSint(_command.EmitterID[0]);
// add command.EmitterID[1]
CreateCommandPayload.AddSint(_command.EmitterID[1]);
// add command.EmitterID[2]
CreateCommandPayload.AddSint(_command.EmitterID[2]);
// add command.EmitterID[3]
CreateCommandPayload.AddSint(_command.EmitterID[3]);
// add command.ListenerID
CreateCommandPayload.AddSint(_command.ListenerID);
// add command.Reserve
CreateCommandPayload.AddByte(_command.Reserve);

// Create logging
CreateCommandPayloadLog(AxesGroup := AxesGroup);
END_METHOD

METHOD INTERNAL CreateCommandPayloadLog
VAR_IN_OUT
  /// Robot assignment of function
  AxesGroup : AxesGroup; 
END_VAR
VAR 
  /// internal index for loops
 _idx : DINT;
END_VAR
// Create log entry for Parameter start
CreateLogMessage      ( Timestamp   := AxesGroup.InternalData.SystemTime,
                        MessageType := MessageType.CMD,
                        Severity    := Severity.DEBUG,
                        MessageCode := 0,
                        MessageText := 'Create command payload with the following parameter(s) :');
  
// Create log entry for EmitterID[x]
FOR _idx := 0 TO 3
DO
  CreateLogMessagePara2 ( Timestamp   := AxesGroup.InternalData.SystemTime,
                          MessageType := MessageType.CMD,
                          Severity    := Severity.DEBUG,
                          MessageCode := 0,
                          MessageText := 'Command.EmitterID[{2}] = {1}',
                          Para1       :=  SINT_TO_STRING(_command.EmitterID[_idx]),
                          Para2       :=  DINT_TO_STRING(_idx));
END_FOR

// Create log entry for ListenerID
CreateLogMessagePara1 ( Timestamp   := AxesGroup.InternalData.SystemTime,
                        MessageType := MessageType.CMD,
                        Severity    := Severity.DEBUG,
                        MessageCode := 0,
                        MessageText := 'Command.ListenerID = {1}',
                        Para1       :=  SINT_TO_STRING(_command.ListenerID));

// Create log entry for Reserve
CreateLogMessagePara1 ( Timestamp   := AxesGroup.InternalData.SystemTime,
                        MessageType := MessageType.CMD,
                        Severity    := Severity.DEBUG,
                        MessageCode := 0,
                        MessageText := 'Command.Reserve = {1}',
                        Para1       :=  BYTE_TO_STRING(_command.Reserve));
END_METHOD

METHOD FB_init : BOOL
VAR_INPUT
  /// if TRUE, the retain variables are initialized (warm start / cold start)
  bInitRetains : BOOL; 
  /// if TRUE, the instance afterwards gets moved into the copy code (online change)
  bInCopyCode  : BOOL;  
END_VAR
MyType := 'MC_ActivateNextCommandFB';

ExecMode := ExecutionMode.PARALLEL;
END_METHOD

METHOD PROTECTED OnCall
VAR_IN_OUT
  /// Robot assignment of function
  AxesGroup : AxesGroup; 
END_VAR
// call base implementation
SUPER^.OnCall(AxesGroup := AxesGroup);

CASE _stepCmd OF
  
  00:  IF ( _execute_R.Q )  
       THEN
         // Check function is supported and parameter are valid ?
         IF (( CheckFunctionSupported( AxesGroup := AxesGroup )) AND
             ( CheckParameterValid   ( AxesGroup := AxesGroup )))      
         THEN
           // set busy flag
           Busy := TRUE;
           // Reset command outputs
           SysDepMemSet(pDest := ADR(OutCmd), Value := 0, DataLen := SIZEOF(OutCmd));         
           // apply command parameter
          _parCmd := ParCmd;
           // init parameter sequence
          _command.ParSeq := 1;
           // create command data
           CommandData := CreateCommandPayload(AxesGroup := AxesGroup);
           // Add command to active command register
          _uniqueID := AxesGroup.Acyclic.ActiveCommandRegister.AddCmd( pCommandFB := ADR(THIS^ ));     
           // set timeout
           SetTimeout(PT := _timeoutCmd, rTimer := _timerCmd);
           // inc step counter
          _stepCmd := _stepCmd + 1;
         END_IF 
       END_IF


  01:  // Wait for responce received
       IF ( _responseReceived )
       THEN
         // reset response received flag
        _responseReceived := FALSE;

         CASE  _response.State 
         OF
           CmdMessageState.BUFFERED    : CommandBuffered    := TRUE;
           CmdMessageState.DONE        : Done               := TRUE;
         //CmdMessageState.ACTIVE      : Active             := TRUE;
         //CmdMessageState.INTERRUPTED : CommandInterrupted := TRUE;
         //CmdMessageState.ABORTED     : CommandAborted     := TRUE;
           CmdMessageState.ERROR       : Error              := TRUE;
         END_CASE

         // Done, Aborted or Error ?
         IF (_response.State >= CmdMessageState.DONE )
         THEN
           // reset busy flag
           Busy := FALSE;
           // Update results
           OutCmd.InvocationCounter := _response.InvocationCounter;
           OutCmd.OriginID          := _response.OriginID;
           // set timeout
           SetTimeout(PT := _timeoutCmd, rTimer := _timerCmd);
           // inc step counter
          _stepCmd := _stepCmd + 1; 
         END_IF
       END_IF


  02: IF ( NOT Execute)
      THEN
        Reset();
       END_IF     
ELSE
  // invalid step
  ErrorID := RobotLibraryEvents.ERR_INVALID_STEP;
END_CASE


// Reset FB
IF ( NOT Execute )
THEN
  Reset();  
END_IF
END_METHOD

METHOD INTERNAL ParseResponsePayload : DINT
VAR_INPUT
  /// Response data
  ResponseData : RobotLibraryRecvDataFB;
  /// Timestamp
  Timestamp    : SystemTime;  
END_VAR
// Table 6-663: Received CMD payload (RC to PLC) of "ActivateNextCommand"
// --------------------------
// Header
// --------------------------
// Byte 00 : USINT - ParSeq | State     
// Byte 01 : SINT  - AlarmMessageSeverity    
// Byte 02 : UINT  - AlarmMessageCode HB
// Byte 03 :       - AlarmMessageCode LB
// --------------------------
// Datablock
// --------------------------
// Byte 04 : USINT - InvocationCounter
// Byte 05 : SINT  - Reserved
// Byte 06 : INT   - OriginID HB
// Byte 07 : INT   - OriginID LB
// --------------------------
// call base implementation to parse the header from payload buffer
ResponseData.PayloadPtr := SUPER^.ParseResponsePayload(ResponseData := ResponseData, Timestamp := Timestamp);

// copy parsed header to response
_response.ParSeq               := _rspHeader.ParSeq;
_response.State                := _rspHeader.State;
_response.AlarmMessageSeverity := _rspHeader.AlarmMessageSeverity;
_response.AlarmMessageCode     := _rspHeader.AlarmMessageCode;

// Get InvocationCounter
_response.InvocationCounter    := ResponseData.GetUsint();
// Get Reserve
_response.Reserve              := ResponseData.GetSint();
// Get OriginID
_response.OriginID             := ResponseData.GetInt();


// Create logging
ParseResponsePayloadLog(ResponseData := ResponseData, Timestamp := Timestamp);
END_METHOD

METHOD INTERNAL ParseResponsePayloadLog
VAR_INPUT
  /// Response data
  ResponseData : RobotLibraryRecvDataFB;
  /// Timestamp
  Timestamp    : SystemTime;  
END_VAR
// Create log entry for Parameter start
CreateLogMessage      ( Timestamp   := Timestamp,
                        MessageType := MessageType.CMD,
                        Severity    := Severity.DEBUG,
                        MessageCode := 0,
                        MessageText := 'Parsed the following parameter(s) from response data:');
                        
// Create log entry for InvocationCounter
CreateLogMessagePara1 ( Timestamp   := Timestamp,
                        MessageType := MessageType.CMD,
                        Severity    := Severity.DEBUG,
                        MessageCode := 0,
                        MessageText := 'Response.InvocationCounter = {1}',
                        Para1       :=  USINT_TO_STRING(_response.InvocationCounter));

// Create log entry for Reserve
CreateLogMessagePara1 ( Timestamp   := Timestamp,
                        MessageType := MessageType.CMD,
                        Severity    := Severity.DEBUG,
                        MessageCode := 0,
                        MessageText := 'Response.Reserve = {1}',
                        Para1       :=  SINT_TO_STRING(_response.Reserve));

// Create log entry for OriginID
CreateLogMessagePara1 ( Timestamp   := Timestamp,
                        MessageType := MessageType.CMD,
                        Severity    := Severity.DEBUG,
                        MessageCode := 0,
                        MessageText := 'Response.OriginID = {1}',
                        Para1       :=  INT_TO_STRING(_response.OriginID));
END_METHOD

METHOD PROTECTED Reset : DINT
VAR_INPUT
END_VAR
Reset := SUPER^.Reset();

Done            := FALSE;
Busy            := FALSE;
CommandBuffered := FALSE;
END_METHOD

END_FUNCTION_BLOCK

// Library/POUs/Additional/MC_AvoidSingularity/MC_AvoidSingularityFB
/// Activate/Deactivate functionality to avoid singularities
FUNCTION_BLOCK MC_AvoidSingularityFB EXTENDS RobotLibraryBaseEnableFB
// ------------------------------------------------------------------------- 
//  SRCI Robot Library                                                
// ------------------------------------------------------------------------- 
//                                                                           
//  Object:      AvoidSingularityFB                                       
//  Author:      Thorsten Brach                                                
//  Date:        2024-06-01
//
//  Description:                                              
//   
//                                                                           
//  Copyright: 
//    (C) 2024 Thorsten Brach. All rights reserved                                                                                                                                            
//             Licensed under the LGPL-3.0 license.
//                                                                           
//  Disclaimer:                                                                           
//    This project is provided without any guarantee and can be used for   
//    private and commercial purposes. Any use is at the user’s 
//    own risk and responsibility.
//
// -------------------------------------------------------------------------
VAR_INPUT
  /// Command parameter 
  ParCmd            : AvoidSingularityParCmd;
END_VAR

VAR_OUTPUT
  /// Command is transferred and confirmed by the RC
  CommandBuffered   : BOOL;
  /// Receiving of input parameter values has been acknowledged by RC
  ParameterAccepted : BOOL;
  /// command results
  OutCmd            : AvoidSingularityOutCmd;  
END_VAR


VAR
  /// internal copy of command parameter 
 _parCmd            : AvoidSingularityParCmd;
  /// command data to send
 _command           : AvoidSingularitySendData;
  /// response data received
 _response          : AvoidSingularityRecvData;
END_VAR

SUPER^(AxesGroup := AxesGroup);

METHOD PROTECTED CheckFunctionSupported : BOOL
VAR_IN_OUT
  /// Robot assignment of function
  AxesGroup : AxesGroup; 
END_VAR
CheckFunctionSupported := AxesGroup.InternalData.RCSupportedFunctions.AvoidSingularity;

IF ( NOT CheckFunctionSupported )
THEN
  // call base implementation for set error and create log entry
  SUPER^.CheckFunctionSupported(AxesGroup := AxesGroup);
END_IF
END_METHOD

METHOD PROTECTED CheckParameterChanged : BOOL
VAR_IN_OUT
  /// Robot assignment of function
  AxesGroup    : AxesGroup; 
END_VAR
// Check ParCmd Size is > 0, because MemCmp does not work correctly with size = 0
IF (SIZEOF(ParCmd) = 0) 
THEN 
  RETURN;
END_IF

// compare memory 
_parameterChanged := ( SysDepMemCmp(pData1 := ADR(ParCmd), pData2 := ADR(_parCmd), DataLen := SIZEOF(ParCmd)) <> RobotLibraryConstants.OK );

// check parameter valid ?
_parameterValid   := CheckParameterValid( AxesGroup := AxesGroup );

IF ((  _parameterChanged        )  AND 
    (  _parameterValid          )) OR
    (  _parameterUpdateInternal )  
THEN  
  // reset internal flag for send parameter update
 _parameterUpdateInternal := FALSE;
  // update internal copy of parameters 
 _parCmd := ParCmd;
  // inc parameter sequence
 _command.ParSeq := _command.ParSeq + 1;
  // update command data  
  CommandData := CreateCommandPayload(AxesGroup := AxesGroup); // ( Access via reference to rCommandFB in ACR )
  // notify active command register 
  AxesGroup.Acyclic.ActiveCommandRegister.NotifyParameterChanged := _uniqueID;  
  // Reset parameter accepted flag
  ParameterAccepted := FALSE;
END_IF
END_METHOD

METHOD INTERNAL CreateCommandPayload : RobotLibrarySendDataFB
VAR_IN_OUT
  /// Robot assignment of function
  AxesGroup : AxesGroup; 
END_VAR
// Table 6-709: Sent CMD payload (PLC to RC) of "AvoidSingularity"
// --------------------------
// Header
// --------------------------
// Byte 00 : UINT  - Type HB     
// Byte 01 :       - Type LB    
// Byte 02 : USINT - Reserve | ExecutionMode
// Byte 03 : USINT - ParSeq  | Priority
// --------------------------
// Datablock
// --------------------------
// Byte 04 : BOOL   - Enable
// Byte 05 : USINT  - Mode
// --------------------------
// set command parameter 
_command.CmdTyp    :=  CmdType.AvoidSingularity;
_command.ExecMode  :=  ExecMode;
_command.ParSeq    := _command.ParSeq;
_command.Priority  :=  Priority;
_command.Enable    :=  Enable;
_command.Mode      := _parCmd.Mode;

// copy command data to header
_cmdHeader := _command;
// call base implementation to copy header to payload buffer
CreateCommandPayload := SUPER^.CreateCommandPayload(AxesGroup := AxesGroup);

// add command.Enable
CreateCommandPayload.AddBool(_command.Enable);
// add command.Mode
CreateCommandPayload.AddByte(_command.Mode);


// Create logging
CreateCommandPayloadLog(AxesGroup := AxesGroup);
END_METHOD

METHOD INTERNAL CreateCommandPayloadLog
VAR_IN_OUT
  /// Robot assignment of function
  AxesGroup : AxesGroup; 
END_VAR
// Create log entry for Parameter start
CreateLogMessage      ( Timestamp   := AxesGroup.InternalData.SystemTime,
                        MessageType := MessageType.CMD,
                        Severity    := Severity.DEBUG,
                        MessageCode := 0,
                        MessageText := 'Create command payload with the following parameter(s) :');
  
// Create log entry for Enable
CreateLogMessagePara1 ( Timestamp   := AxesGroup.InternalData.SystemTime,
                        MessageType := MessageType.CMD,
                        Severity    := Severity.DEBUG,
                        MessageCode := 0,
                        MessageText := 'Command.Enable = {1}',
                        Para1       :=  BOOL_TO_STRING(_command.Enable));

// Create log entry for Mode
CreateLogMessagePara1 ( Timestamp   := AxesGroup.InternalData.SystemTime,
                        MessageType := MessageType.CMD,
                        Severity    := Severity.DEBUG,
                        MessageCode := 0,
                        MessageText := 'Command.Mode = {1}',
                        Para1       :=  SINGULARITY_AVOIDANCE_MODE_TO_STRING(_command.Mode));
END_METHOD

METHOD FB_init : BOOL
VAR_INPUT
  /// if TRUE, the retain variables are initialized (warm start / cold start)
  bInitRetains : BOOL; 
  /// if TRUE, the instance afterwards gets moved into the copy code (online change)
  bInCopyCode  : BOOL;  
END_VAR
MyType := 'MC_AvoidSingularityFB';

ExecMode := ExecutionMode.PARALLEL;
END_METHOD

METHOD PROTECTED OnCall
VAR_IN_OUT
  /// Robot assignment of function
  AxesGroup : AxesGroup; 
END_VAR
// call base implementation
SUPER^.OnCall(AxesGroup := AxesGroup);

CASE _stepCmd OF
  
  00:  IF ( _enable_R.Q )
       THEN
         // Check function is supported and parameter are valid ?
         IF (( CheckFunctionSupported( AxesGroup := AxesGroup )) AND
             ( CheckParameterValid   ( AxesGroup := AxesGroup )))      
         THEN
           // reset the rising edge
          _enable_R();       
           // reset the falling edge
          _enable_F();       
           // set busy flag
           Busy := TRUE;
           // Reset command outputs
           SysDepMemSet(pDest := ADR(OutCmd), Value := 0, DataLen := SIZEOF(OutCmd));         
           // apply command parameter
          _parCmd := ParCmd;
           // init parameter sequence
          _command.ParSeq := 1;
           // create command data
           CommandData := CreateCommandPayload(AxesGroup := AxesGroup);
           // Add command to active command register
          _uniqueID := AxesGroup.Acyclic.ActiveCommandRegister.AddCmd( pCommandFB := ADR(THIS^ ));     
           // set timeout
           SetTimeout(PT := _timeoutCmd, rTimer := _timerCmd);
           // inc step counter
          _stepCmd := _stepCmd + 1; 
         END_IF
       END_IF     


  01:  // Wait for responce received
       IF ( _responseReceived )
       THEN
         // reset response received flag
        _responseReceived := FALSE;

         CASE  _response.State 
         OF
           CmdMessageState.BUFFERED    : CommandBuffered    := TRUE;
           CmdMessageState.ACTIVE      : ParameterAccepted  := TRUE;           
           CmdMessageState.ERROR       : Error              := TRUE;
         END_CASE
         
         // Update results
         Enabled := _response.Enabled;
                
         // Done, Aborted or Error ?
         IF (_response.State >= CmdMessageState.DONE )
         THEN
           // Reset enabled flag
           Enabled := FALSE;
           // set timeout
           SetTimeout(PT := _timeoutCmd, rTimer := _timerCmd);
           // inc step counter
          _stepCmd := _stepCmd + 1; 
         END_IF
       END_IF
       
       // do not abort directly, so that the ParSeq update can be send
       IF ( _enable_R.Q ) OR ( _enable_F.Q ) 
       THEN
         // trigger parameter update to disable FB
        _parameterUpdateInternal := TRUE;
         // reset the rising edge
        _enable_R();       
         // reset the falling edge
        _enable_F();       
       END_IF


  02: IF (NOT Enable)
      THEN
        Reset();   
      END_IF
ELSE
  // invalid step
  ErrorID := RobotLibraryEvents.ERR_INVALID_STEP;
END_CASE



// Reset FB
IF (( _enable_R.Q ) OR
    ( _enable_F.Q ))
THEN
  Reset(); 
END_IF
END_METHOD

METHOD INTERNAL ParseResponsePayload : DINT
VAR_INPUT
  /// Response data
  ResponseData : RobotLibraryRecvDataFB;
  /// Timestamp
  Timestamp    : SystemTime;  
END_VAR
// Table 6-710: Received CMD payload (RC to PLC) of "AvoidSingularity"
// --------------------------
// Header
// --------------------------
// Byte 00 : USINT - ParSeq | State     
// Byte 01 : SINT  - AlarmMessageSeverity    
// Byte 02 : UINT  - AlarmMessageCode HB
// Byte 03 :       - AlarmMessageCode LB
// --------------------------
// Datablock
// --------------------------
// Byte 04 : BOOL  - Enabled
// --------------------------
// call base implementation to parse the header from payload buffer
ResponseData.PayloadPtr := SUPER^.ParseResponsePayload(ResponseData := ResponseData, Timestamp := Timestamp);

// copy parsed header to response
_response.ParSeq               := _rspHeader.ParSeq;
_response.State                := _rspHeader.State;
_response.AlarmMessageSeverity := _rspHeader.AlarmMessageSeverity;
_response.AlarmMessageCode     := _rspHeader.AlarmMessageCode;

// Get Response.Enabled
_response.Enabled := ResponseData.GetBool();


// Create logging
ParseResponsePayloadLog(ResponseData := ResponseData, Timestamp := Timestamp);
END_METHOD

METHOD INTERNAL ParseResponsePayloadLog
VAR_INPUT
  /// Response data
  ResponseData : RobotLibraryRecvDataFB;
  /// Timestamp
  Timestamp    : SystemTime;  
END_VAR
// Create log entry for Parameter start
CreateLogMessage      ( Timestamp   := Timestamp,
                        MessageType := MessageType.CMD,
                        Severity    := Severity.DEBUG,
                        MessageCode := 0,
                        MessageText := 'Parsed the following parameter(s) from response data:');
                        
// Create log entry for Enabled
CreateLogMessagePara1 ( Timestamp   := Timestamp,
                        MessageType := MessageType.CMD,
                        Severity    := Severity.DEBUG,
                        MessageCode := 0,
                        MessageText := 'Response.Enabled = {1}',
                        Para1       :=  BOOL_TO_STRING(_response.Enabled));
END_METHOD

METHOD PROTECTED Reset : DINT
VAR_INPUT
END_VAR
Reset := SUPER^.Reset();

Busy               := FALSE;
CommandBuffered    := FALSE;
END_METHOD

END_FUNCTION_BLOCK

// Library/POUs/Additional/MC_BrakeTest/MC_BrakeTestFB
/// Activate robot cycle brake test and give feedback to PLC
FUNCTION_BLOCK MC_BrakeTestFB EXTENDS RobotLibraryBaseExecuteFB
// ------------------------------------------------------------------------- 
//  SRCI Robot Library                                                
// ------------------------------------------------------------------------- 
//                                                                           
//  Object:      BrakeTest                                       
//  Author:      Thorsten Brach                                                
//  Date:        2024-06-01
//
//  Description:                                              
//   
//                                                                           
//  Copyright: 
//    (C) 2024 Thorsten Brach. All rights reserved                                                                                                                                            
//             Licensed under the LGPL-3.0 license.
//                                                                           
//  Disclaimer:                                                                           
//    This project is provided without any guarantee and can be used for   
//    private and commercial purposes. Any use is at the user’s 
//    own risk and responsibility.
//
// -------------------------------------------------------------------------
VAR_INPUT
  /// Command parameter 
  ParCmd             : BrakeTestParCmd;
END_VAR
VAR_OUTPUT
  /// Command is transferred and confirmed by the RC
  CommandBuffered    : BOOL;
  /// During the realization of the brake test, the command controls the motion of the respective axis group.
  /// TRUE: The brake test is being realized
  /// FALSE: The brake test is not realized
  Active             : BOOL;
  /// The command was aborted by another command.
  CommandAborted     : BOOL;
  /// TRUE, while command is interrupted during execution and can be continued
  CommandInterrupted : BOOL; 
  /// Command output 
  OutCmd             : BrakeTestOutCmd;
END_VAR

var
  /// internal copy of command parameter 
 _parCmd             : BrakeTestParCmd;
  /// command data to send
 _command            : BrakeTestSendData;
  /// response data received
 _response           : BrakeTestRecvData;      
END_VAR

SUPER^(AxesGroup := AxesGroup);

METHOD PROTECTED CheckFunctionSupported : BOOL
VAR_IN_OUT
  /// Robot assignment of function
  AxesGroup : AxesGroup; 
END_VAR
CheckFunctionSupported := AxesGroup.InternalData.RCSupportedFunctions.BrakeTest;

IF ( NOT CheckFunctionSupported )
THEN
  // call base implementation for set error and create log entry
  SUPER^.CheckFunctionSupported(AxesGroup := AxesGroup);
END_IF
END_METHOD

METHOD PROTECTED CheckParameterChanged : BOOL
VAR_IN_OUT
  /// Robot assignment of function
  AxesGroup    : AxesGroup; 
END_VAR
// Check ParCmd Size is > 0, because MemCmp does not work correctly with size = 0
IF (SIZEOF(ParCmd) = 0) 
THEN 
  RETURN;
END_IF

// compare memory 
_parameterChanged := ( SysDepMemCmp(pData1 := ADR(ParCmd), pData2 := ADR(_parCmd), DataLen := SIZEOF(ParCmd)) <> RobotLibraryConstants.OK );

// check parameter valid ?
_parameterValid   := CheckParameterValid( AxesGroup := AxesGroup );

IF ((  _parameterChanged        )  AND 
    (  _parameterValid          )) OR
    (  _parameterUpdateInternal )  
THEN  
  // reset internal flag for send parameter update
 _parameterUpdateInternal := FALSE;
  // update internal copy of parameters 
 _parCmd := ParCmd;
  // inc parameter sequence
 _command.ParSeq := _command.ParSeq + 1;
  // update command data  
  CommandData := CreateCommandPayload(AxesGroup := AxesGroup); // ( Access via reference to rCommandFB in ACR )
  // notify active command register 
  AxesGroup.Acyclic.ActiveCommandRegister.NotifyParameterChanged := _uniqueID;  
END_IF
END_METHOD

METHOD INTERNAL CreateCommandPayload : RobotLibrarySendDataFB
VAR_IN_OUT
  /// Robot assignment of function
  AxesGroup : AxesGroup; 
END_VAR
// Table 6-740: Sent CMD payload (PLC to RC) of "BrakeTest"
// --------------------------
// Header
// --------------------------
// Byte 00 : UINT  - Type HB     
// Byte 01 :       - Type LB    
// Byte 02 : USINT - Reserve | ExecutionMode
// Byte 03 : USINT - ParSeq  | Priority
// --------------------------
// Datablock
// --------------------------
// Byte 04 : BYTE - RobotAxesActive
// Byte 05 : BYTE - ExternalAxesActive
// --------------------------
// set command parameter 
_command.CmdTyp               :=  CmdType.BrakeTest;
_command.ExecMode             :=  ExecMode;
_command.ParSeq               := _command.ParSeq;
_command.Priority             :=  Priority;
_command.RobotAxesActive.0    := _parCmd.RobotAxesActive.Bit00;
_command.RobotAxesActive.1    := _parCmd.RobotAxesActive.AxisJ1;
_command.RobotAxesActive.2    := _parCmd.RobotAxesActive.AxisJ2;
_command.RobotAxesActive.3    := _parCmd.RobotAxesActive.AxisJ3;
_command.RobotAxesActive.4    := _parCmd.RobotAxesActive.AxisJ4;
_command.RobotAxesActive.5    := _parCmd.RobotAxesActive.AxisJ5;
_command.RobotAxesActive.6    := _parCmd.RobotAxesActive.AxisJ6;
_command.RobotAxesActive.7    := _parCmd.RobotAxesActive.Bit07;
_command.ExternalAxesActive.0 := _parCmd.ExternalAxesActive.Bit00;
_command.ExternalAxesActive.1 := _parCmd.ExternalAxesActive.AxisE1;
_command.ExternalAxesActive.2 := _parCmd.ExternalAxesActive.AxisE2;
_command.ExternalAxesActive.3 := _parCmd.ExternalAxesActive.AxisE3;
_command.ExternalAxesActive.4 := _parCmd.ExternalAxesActive.AxisE4;
_command.ExternalAxesActive.5 := _parCmd.ExternalAxesActive.AxisE5;
_command.ExternalAxesActive.6 := _parCmd.ExternalAxesActive.AxisE6;
_command.ExternalAxesActive.7 := _parCmd.ExternalAxesActive.Bit07;

// copy command data to header
_cmdHeader := _command;
// call base implementation to copy header to payload buffer
CreateCommandPayload := SUPER^.CreateCommandPayload(AxesGroup := AxesGroup);

// add command.EmitterID[0]
CreateCommandPayload.AddByte(_command.RobotAxesActive);
// add command.EmitterID[1]
CreateCommandPayload.AddByte(_command.ExternalAxesActive);


// Create logging
CreateCommandPayloadLog(AxesGroup := AxesGroup);
END_METHOD

METHOD INTERNAL CreateCommandPayloadLog
VAR_IN_OUT
  /// Robot assignment of function
  AxesGroup : AxesGroup; 
END_VAR
// Create log entry for Parameter start
CreateLogMessage      ( Timestamp   := AxesGroup.InternalData.SystemTime,
                        MessageType := MessageType.CMD,
                        Severity    := Severity.DEBUG,
                        MessageCode := 0,
                        MessageText := 'Create command payload with the following parameter(s) :');
  
// Create log entry for RobotAxesActive
CreateLogMessagePara1 ( Timestamp   := AxesGroup.InternalData.SystemTime,
                        MessageType := MessageType.CMD,
                        Severity    := Severity.DEBUG,
                        MessageCode := 0,
                        MessageText := 'Command.RobotAxesActive = {1}',
                        Para1       :=  BYTE_TO_STRING_BIN(_command.RobotAxesActive));

// Create log entry for ExternalAxesActive
CreateLogMessagePara1 ( Timestamp   := AxesGroup.InternalData.SystemTime,
                        MessageType := MessageType.CMD,
                        Severity    := Severity.DEBUG,
                        MessageCode := 0,
                        MessageText := 'Command.ExternalAxesActive = {1}',
                        Para1       :=  BYTE_TO_STRING_BIN(_command.ExternalAxesActive));
END_METHOD

METHOD FB_init : BOOL
VAR_INPUT
  /// if TRUE, the retain variables are initialized (warm start / cold start)
  bInitRetains : BOOL; 
  /// if TRUE, the instance afterwards gets moved into the copy code (online change)
  bInCopyCode  : BOOL;  
END_VAR
MyType := 'MC_BrakeTestFB';
END_METHOD

METHOD PROTECTED OnCall
VAR_IN_OUT
  /// Robot assignment of function
  AxesGroup : AxesGroup; 
END_VAR
// call base implementation
SUPER^.OnCall(AxesGroup := AxesGroup);

CASE _stepCmd OF
  
  00:  IF ( _execute_R.Q ) 
       THEN
         // Check function is supported and parameter are valid ?
         IF (( CheckFunctionSupported( AxesGroup := AxesGroup )) AND
             ( CheckParameterValid   ( AxesGroup := AxesGroup )))      
         THEN
           // set busy flag
           Busy := TRUE;
           // Reset command outputs
           SysDepMemSet(pDest := ADR(OutCmd), Value := 0, DataLen := SIZEOF(OutCmd));         
           // apply command parameter
          _parCmd := ParCmd;
           // init parameter sequence
          _command.ParSeq := 1;
           // create command data
           CommandData := CreateCommandPayload(AxesGroup := AxesGroup);
           // Add command to active command register
          _uniqueID := AxesGroup.Acyclic.ActiveCommandRegister.AddCmd( pCommandFB := ADR(THIS^ ));     
           // set timeout
           SetTimeout(PT := _timeoutCmd, rTimer := _timerCmd);
           // inc step counter
          _stepCmd := _stepCmd + 1;
         END_IF 
       END_IF
     

  01:  // Wait for responce received
       IF ( _responseReceived )
       THEN
         // reset response received flag
        _responseReceived := FALSE;
         // reset Active flag
         Active := FALSE;
         
         CASE  _response.State 
         OF
           CmdMessageState.BUFFERED    : CommandBuffered    := TRUE;
           CmdMessageState.ACTIVE      : Active             := TRUE;
           CmdMessageState.INTERRUPTED : CommandInterrupted := TRUE;
           CmdMessageState.DONE        : Done               := TRUE;
           CmdMessageState.ABORTED     : CommandAborted     := TRUE;
           CmdMessageState.ERROR       : Error              := TRUE;
         END_CASE
                
         // Done, Aborted or Error ?
         IF (_response.State >= CmdMessageState.DONE )
         THEN 
           // reset busy flag          
           Busy := FALSE;
           // Update results
           OutCmd.RobotAxesStatus.Bit00     := _response.RobotAxesStatus.0;
           OutCmd.RobotAxesStatus.AxisJ1    := _response.RobotAxesStatus.1;
           OutCmd.RobotAxesStatus.AxisJ2    := _response.RobotAxesStatus.2;
           OutCmd.RobotAxesStatus.AxisJ3    := _response.RobotAxesStatus.3;
           OutCmd.RobotAxesStatus.AxisJ4    := _response.RobotAxesStatus.4;
           OutCmd.RobotAxesStatus.AxisJ5    := _response.RobotAxesStatus.5;
           OutCmd.RobotAxesStatus.AxisJ6    := _response.RobotAxesStatus.6;
           OutCmd.RobotAxesStatus.Bit07     := _response.RobotAxesStatus.7;
           
           OutCmd.RobotAxesWarning.Bit00     := _response.RobotAxesWarning.0;
           OutCmd.RobotAxesWarning.AxisJ1    := _response.RobotAxesWarning.1;
           OutCmd.RobotAxesWarning.AxisJ2    := _response.RobotAxesWarning.2;
           OutCmd.RobotAxesWarning.AxisJ3    := _response.RobotAxesWarning.3;
           OutCmd.RobotAxesWarning.AxisJ4    := _response.RobotAxesWarning.4;
           OutCmd.RobotAxesWarning.AxisJ5    := _response.RobotAxesWarning.5;
           OutCmd.RobotAxesWarning.AxisJ6    := _response.RobotAxesWarning.6;
           OutCmd.RobotAxesWarning.Bit07     := _response.RobotAxesWarning.7;

           OutCmd.ExternalAxesStatus.Bit00   := _response.ExternalAxesStatus.0;
           OutCmd.ExternalAxesStatus.AxisE1  := _response.ExternalAxesStatus.1;
           OutCmd.ExternalAxesStatus.AxisE2  := _response.ExternalAxesStatus.2;
           OutCmd.ExternalAxesStatus.AxisE3  := _response.ExternalAxesStatus.3;
           OutCmd.ExternalAxesStatus.AxisE4  := _response.ExternalAxesStatus.4;
           OutCmd.ExternalAxesStatus.AxisE5  := _response.ExternalAxesStatus.5;
           OutCmd.ExternalAxesStatus.AxisE6  := _response.ExternalAxesStatus.6;
           OutCmd.ExternalAxesStatus.Bit07   := _response.ExternalAxesStatus.7;

           OutCmd.ExternalAxesWarning.Bit00  := _response.ExternalAxesWarning.0;
           OutCmd.ExternalAxesWarning.AxisE1 := _response.ExternalAxesWarning.1;
           OutCmd.ExternalAxesWarning.AxisE2 := _response.ExternalAxesWarning.2;
           OutCmd.ExternalAxesWarning.AxisE3 := _response.ExternalAxesWarning.3;
           OutCmd.ExternalAxesWarning.AxisE4 := _response.ExternalAxesWarning.4;
           OutCmd.ExternalAxesWarning.AxisE5 := _response.ExternalAxesWarning.5;
           OutCmd.ExternalAxesWarning.AxisE6 := _response.ExternalAxesWarning.6;
           OutCmd.ExternalAxesWarning.Bit07  := _response.ExternalAxesWarning.7;
           
           // set timeout
           SetTimeout(PT := _timeoutCmd, rTimer := _timerCmd);
           // inc step counter
          _stepCmd := _stepCmd + 1; 
         END_IF
       END_IF

  02: IF ( NOT Execute)
      THEN
        Reset();
      END_IF     
ELSE
  // invalid step
  ErrorID := RobotLibraryEvents.ERR_INVALID_STEP;
END_CASE


// Reset FB
IF ( NOT Execute )
THEN
  Reset();  
END_IF
END_METHOD

METHOD INTERNAL ParseResponsePayload : DINT
VAR_INPUT
  /// Response data
  ResponseData : RobotLibraryRecvDataFB;
  /// Timestamp
  Timestamp    : SystemTime;  
END_VAR
// Table 6-741: Received CMD payload (RC to PLC) of "BrakeTest"
// --------------------------
// Header
// --------------------------
// Byte 00 : USINT - ParSeq | State     
// Byte 01 : SINT  - AlarmMessageSeverity    
// Byte 02 : UINT  - AlarmMessageCode HB
// Byte 03 :       - AlarmMessageCode LB
// --------------------------
// Datablock
// --------------------------
// Byte 04 : BYTE  - RobotAxesStatus
// Byte 05 : BYTE  - ExternalAxesStatus
// Byte 06 : BYTE  - RobotAxesWarning
// Byte 07 : BYTE  - ExternalAxesWarning
// --------------------------
// call base implementation to parse the header from payload buffer
ResponseData.PayloadPtr := SUPER^.ParseResponsePayload(ResponseData := ResponseData, Timestamp := Timestamp);

// copy parsed header to response
_response.ParSeq               := _rspHeader.ParSeq;
_response.State                := _rspHeader.State;
_response.AlarmMessageSeverity := _rspHeader.AlarmMessageSeverity;
_response.AlarmMessageCode     := _rspHeader.AlarmMessageCode;

// Get RobotAxesStatus
_response.RobotAxesStatus     := ResponseData.GetByte();
// Get ExternalAxesStatus
_response.ExternalAxesStatus  := ResponseData.GetByte();
// Get RobotAxesWarning
_response.RobotAxesWarning    := ResponseData.GetByte();
// Get ExternalAxesWarning
_response.ExternalAxesWarning := ResponseData.GetByte();

// Create logging
ParseResponsePayloadLog(ResponseData := ResponseData, Timestamp := Timestamp);
END_METHOD

METHOD INTERNAL ParseResponsePayloadLog
VAR_INPUT
  /// Response data
  ResponseData : RobotLibraryRecvDataFB;
  /// Timestamp
  Timestamp    : SystemTime;  
END_VAR
// Create log entry for Parameter start
CreateLogMessage      ( Timestamp   := Timestamp,
                        MessageType := MessageType.CMD,
                        Severity    := Severity.DEBUG,
                        MessageCode := 0,
                        MessageText := 'Parsed the following parameter(s) from response data:');
                        
// Create log entry for RobotAxesStatus
CreateLogMessagePara1 ( Timestamp   := Timestamp,
                        MessageType := MessageType.CMD,
                        Severity    := Severity.DEBUG,
                        MessageCode := 0,
                        MessageText := 'Response.RobotAxesStatus = {1}',
                        Para1       :=  BYTE_TO_STRING_BIN(_response.RobotAxesStatus));

// Create log entry for ExternalAxesStatus
CreateLogMessagePara1 ( Timestamp   := Timestamp,
                        MessageType := MessageType.CMD,
                        Severity    := Severity.DEBUG,
                        MessageCode := 0,
                        MessageText := 'Response.ExternalAxesStatus = {1}',
                        Para1       :=  BYTE_TO_STRING_BIN(_response.ExternalAxesStatus));

// Create log entry for RobotAxesWarning
CreateLogMessagePara1 ( Timestamp   := Timestamp,
                        MessageType := MessageType.CMD,
                        Severity    := Severity.DEBUG,
                        MessageCode := 0,
                        MessageText := 'Response.RobotAxesWarning = {1}',
                        Para1       :=  BYTE_TO_STRING_BIN(_response.RobotAxesWarning));

// Create log entry for ExternalAxesWarning
CreateLogMessagePara1 ( Timestamp   := Timestamp,
                        MessageType := MessageType.CMD,
                        Severity    := Severity.DEBUG,
                        MessageCode := 0,
                        MessageText := 'Response.ExternalAxesWarning = {1}',
                        Para1       :=  BYTE_TO_STRING_BIN(_response.ExternalAxesWarning));
END_METHOD

METHOD PROTECTED Reset : DINT
VAR_INPUT
END_VAR
Reset := SUPER^.Reset();

Done               := FALSE;
Busy               := FALSE;
Active             := FALSE;
CommandBuffered    := FALSE;
CommandAborted     := FALSE;
CommandInterrupted := FALSE;
END_METHOD

END_FUNCTION_BLOCK

// Library/POUs/Additional/MC_CallSubprogram/MC_CallSubprogramFB
/// Call subprogram stored in RC from PLC
FUNCTION_BLOCK MC_CallSubprogramFB EXTENDS RobotLibraryBaseExecuteFB
// ------------------------------------------------------------------------- 
//  SRCI Robot Library                                                
// ------------------------------------------------------------------------- 
//                                                                           
//  Object:      CallSubprogramFB                                       
//  Author:      Thorsten Brach                                                
//  Date:        2024-06-01
//
//  Description:                                              
//   
//                                                                           
//  Copyright: 
//    (C) 2024 Thorsten Brach. All rights reserved                                                                                                                                            
//             Licensed under the LGPL-3.0 license.
//                                                                           
//  Disclaimer:                                                                           
//    This project is provided without any guarantee and can be used for   
//    private and commercial purposes. Any use is at the user’s 
//    own risk and responsibility.
//
// -------------------------------------------------------------------------
VAR_INPUT
  /// command parameter 
  ParCmd             : CallSubprogramParCmd;
  /// Processing mode
  ProcessingMode     : ProcessingMode;
  /// Defines the target sequence in which the command will be executed
  SequenceFlag       : SequenceFlag;
END_VAR

VAR_OUTPUT
  /// TRUE while the output ReturnData returns valid data according to the user defined subprogram
  Valid              : BOOL;
  /// Command is transferred and confirmed by the RC
  CommandBuffered    : BOOL;
  /// The requested subprogram on the RC is in progress. Movement of the axes trough this subprogram is possible.  
  InProgress         : BOOL;
  /// The command was aborted by another command
  CommandAborted     : BOOL;
  /// TRUE, while command is interrupted during execution and can be continued.
  CommandInterrupted : BOOL;
  /// Receiving of input parameter values has been acknowledged by RC
  ParameterAccepted  : BOOL;
  /// command outputs
  OutCmd             : CallSubprogramOutCmd;       
END_VAR



VAR
  /// internal copy of command parameter 
 _parCmd             : CallSubprogramParCmd;
  /// command data to send
 _command            : CallSubprogramSendData;
  /// response data received
 _response           : CallSubprogramRecvData;      
END_VAR

SUPER^(AxesGroup := AxesGroup);

METHOD PROTECTED CheckFunctionSupported : BOOL
VAR_IN_OUT
  /// Robot assignment of function
  AxesGroup : AxesGroup; 
END_VAR
CheckFunctionSupported := AxesGroup.InternalData.RCSupportedFunctions.CallSubprogram;

IF ( NOT CheckFunctionSupported )
THEN
  // call base implementation for set error and create log entry
  SUPER^.CheckFunctionSupported(AxesGroup := AxesGroup);
END_IF
END_METHOD

METHOD PROTECTED CheckParameterChanged : BOOL
VAR_IN_OUT
  /// Robot assignment of function
  AxesGroup    : AxesGroup; 
END_VAR
// Check ParCmd Size is > 0, because MemCmp does not work correctly with size = 0
IF (SIZEOF(ParCmd) = 0) 
THEN 
  RETURN;
END_IF

// compare memory 
_parameterChanged := ( SysDepMemCmp(pData1 := ADR(ParCmd), pData2 := ADR(_parCmd), DataLen := SIZEOF(ParCmd)) <> RobotLibraryConstants.OK );

// check parameter valid ?
_parameterValid   := CheckParameterValid( AxesGroup := AxesGroup );

IF ((  _parameterChanged        )  AND 
    (  _parameterValid          )) OR
    (  _parameterUpdateInternal )  
THEN  
  // reset internal flag for send parameter update
 _parameterUpdateInternal := FALSE;
  // update internal copy of parameters 
 _parCmd := ParCmd;
  // inc parameter sequence
 _command.ParSeq := _command.ParSeq + 1;
  // update command data  
  CommandData := CreateCommandPayload(AxesGroup := AxesGroup); // ( Access via reference to rCommandFB in ACR )
  // notify active command register 
  AxesGroup.Acyclic.ActiveCommandRegister.NotifyParameterChanged := _uniqueID;  
  // Reset parameter accepted flag
  ParameterAccepted := FALSE;
END_IF
END_METHOD

METHOD INTERNAL CreateCommandPayload : RobotLibrarySendDataFB
VAR_IN_OUT
  /// Robot assignment of function
  AxesGroup : AxesGroup; 
END_VAR
// Table 6-687: Sent CMD payload (PLC to RC) of "CallSubprogram"
// --------------------------
// Header
// --------------------------
// Byte 00 : UINT  - Type HB     
// Byte 01 :       - Type LB    
// Byte 02 : USINT - Reserve | ExecutionMode
// Byte 03 : USINT - ParSeq  | Priority
// --------------------------
// Datablock
// --------------------------
// Byte 00 : UINT  Type;
// Byte 01 :       Type;
// Byte 02 : USINT Reserved ExecutionMode;
// Byte 03 : USINT ParSeq Priority;
// Byte 04 : SINT  EmitterID[0];
// Byte 05 : SINT  EmitterID[1];
// Byte 06 : SINT  EmitterID[2];
// Byte 07 : SINT  EmitterID[3];
// Byte 08 : SINT  ListenerID;
// Byte 09 : BYTE  Reserved;
// Byte 10 : UINT  JobID;
// Byte 11 :       JobID;
// Byte 12 : BYTE  Data[0];
// Byte 13 : BYTE  Data[1];
// Byte 14 : BYTE  Data[2];
// Byte 15 : BYTE  Data[3];
// Byte 16 : BYTE  Data[4];
// Byte 17 : BYTE  Data[5];
// Byte 18 : BYTE  Data[6];
// Byte 19 : BYTE  Data[7];
// Byte 20 : BYTE  Data[8];
// Byte 21 : BYTE  Data[9];
// Byte 22 : BYTE  Data[10];
// Byte 23 : BYTE  Data[11];
// Byte 24 : BYTE  Data[12];
// Byte 25 : BYTE  Data[13];
// Byte 26 : BYTE  Data[14];
// Byte 27 : BYTE  Data[15];
// Byte 28 : BYTE  Data[16];
// Byte 29 : BYTE  Data[17];
// Byte 30 : BYTE  Data[18];
// Byte 31 : BYTE  Data[19];
// Byte 32 : BYTE  Data[20];
// Byte 33 : BYTE  Data[21];
// Byte 34 : BYTE  Data[22];
// Byte 35 : BYTE  Data[23];
// Byte 36 : BYTE  Data[24];
// Byte 37 : BYTE  Data[25];
// Byte 38 : BYTE  Data[26];
// Byte 39 : BYTE  Data[27];
// Byte 40 : BYTE  Data[28];
// Byte 41 : BYTE  Data[29];
// Byte 42 : BYTE  Data[30];
// Byte 43 : BYTE  Data[31];
// Byte 44 : BYTE  Data[32];
// Byte 45 : BYTE  Data[33];
// Byte 46 : BYTE  Data[34];
// Byte 47 : BYTE  Data[35];
// Byte 48 : BYTE  Data[36];
// Byte 49 : BYTE  Data[37];
// Byte 50 : BYTE  Data[38];
// Byte 51 : BYTE  Data[39];
// Byte 52 : BYTE  Data[40];
// Byte 53 : BYTE  Data[41];
// Byte 54 : BYTE  Data[42];
// Byte 55 : BYTE  Data[43];
// Byte 56 : BYTE  Data[44];
// Byte 57 : BYTE  Data[45];
// Byte 58 : BYTE  Data[46];
// Byte 59 : BYTE  Data[47];
// Byte 60 : BYTE  Data[48];
// Byte 61 : BYTE  Data[49];
// Byte 62 : BYTE  Data[50];
// Byte 63 : BYTE  Data[51];
// Byte 64 : BYTE  Data[52];
// Byte 65 : BYTE  Data[53];
// Byte 66 : BYTE  Data[54];
// Byte 67 : BYTE  Data[55];
// Byte 68 : BYTE  Data[56];
// Byte 69 : BYTE  Data[57];
// Byte 70 : BYTE  Data[58];
// Byte 71 : BYTE  Data[59];
// Byte 72 : BYTE  Data[60];
// Byte 73 : BYTE  Data[61];
// Byte 74 : BYTE  Data[62];
// Byte 75 : BYTE  Data[63];
// Byte 76 : BYTE  Data[64];
// Byte 77 : BYTE  Data[65];
// Byte 78 : BYTE  Data[66];
// Byte 79 : BYTE  Data[67];
// Byte 80 : BYTE  Data[68];
// Byte 81 : BYTE  Data[69];
// Byte 82 : BYTE  Data[70];
// Byte 83 : BYTE  Data[71];
// Byte 84 : BYTE  Data[72];
// Byte 85 : BYTE  Data[73];
// Byte 86 : BYTE  Data[74];
// Byte 87 : BYTE  Data[75];
// Byte 88 : BYTE  Data[76];
// Byte 89 : BYTE  Data[77];
// Byte 90 : BYTE  Data[78];
// Byte 91 : BYTE  Data[79];
// Byte 92 : BYTE  Data[80];
// Byte 93 : BYTE  Data[81];
// Byte 94 : BYTE  Data[82];
// Byte 95 : BYTE  Data[83];
// Byte 96 : BYTE  Data[84];
// Byte 97 : BYTE  Data[85];
// Byte 98 : BYTE  Data[86];
// Byte 99 : BYTE  Data[87];
// Byte 100: BYTE  Data[88];
// Byte 101: BYTE  Data[89];
// Byte 102: BYTE  Data[90];
// Byte 103: BYTE  Data[91];
// Byte 104: BYTE  Data[92];
// Byte 105: BYTE  Data[93];
// Byte 106: BYTE  Data[94];
// Byte 107: BYTE  Data[95];
// Byte 108: BYTE  Data[96];
// Byte 109: BYTE  Data[97];
// Byte 110: BYTE  Data[98];
// Byte 111: BYTE  Data[99];
// Byte 112: BYTE  Data[100];
// Byte 113: BYTE  Data[101];
// Byte 114: BYTE  Data[102];
// Byte 115: BYTE  Data[103];
// Byte 116: BYTE  Data[104];
// Byte 117: BYTE  Data[105];
// Byte 118: BYTE  Data[106];
// Byte 119: BYTE  Data[107];
// Byte 120: BYTE  Data[108];
// Byte 121: BYTE  Data[109];
// Byte 122: BYTE  Data[110];
// Byte 123: BYTE  Data[111];
// Byte 124: BYTE  Data[112];
// Byte 125: BYTE  Data[113];
// Byte 126: BYTE  Data[114];
// Byte 127: BYTE  Data[115];
// Byte 128: BYTE  Data[116];
// Byte 129: BYTE  Data[117];
// Byte 130: BYTE  Data[118];
// Byte 131: BYTE  Data[119];
// Byte 132: BYTE  Data[120];
// Byte 133: BYTE  Data[121];
// Byte 134: BYTE  Data[122];
// Byte 135: BYTE  Data[123];
// Byte 136: BYTE  Data[124];
// Byte 137: BYTE  Data[125];
// Byte 138: BYTE  Data[126];
// Byte 139: BYTE  Data[127];
// Byte 140: BYTE  Data[128];
// Byte 141: BYTE  Data[129];
// Byte 142: BYTE  Data[130];
// Byte 143: BYTE  Data[131];
// Byte 144: BYTE  Data[132];
// Byte 145: BYTE  Data[133];
// Byte 146: BYTE  Data[134];
// Byte 147: BYTE  Data[135];
// Byte 148: BYTE  Data[136];
// Byte 149: BYTE  Data[137];
// Byte 150: BYTE  Data[138];
// Byte 151: BYTE  Data[139];
// Byte 152: BYTE  Data[140];
// Byte 153: BYTE  Data[141];
// Byte 154: BYTE  Data[142];
// Byte 155: BYTE  Data[143];
// Byte 156: BYTE  Data[144];
// Byte 157: BYTE  Data[145];
// Byte 158: BYTE  Data[146];
// Byte 159: BYTE  Data[147];
// Byte 160: BYTE  Data[148];
// Byte 161: BYTE  Data[149];
// Byte 162: BYTE  Data[150];
// Byte 163: BYTE  Data[151];
// Byte 164: BYTE  Data[152];
// Byte 165: BYTE  Data[153];
// Byte 166: BYTE  Data[154];
// Byte 167: BYTE  Data[155];
// Byte 168: BYTE  Data[156];
// Byte 169: BYTE  Data[157];
// Byte 170: BYTE  Data[158];
// Byte 171: BYTE  Data[159];
// Byte 172: BYTE  Data[160];
// Byte 173: BYTE  Data[161];
// Byte 174: BYTE  Data[162];
// Byte 175: BYTE  Data[163];
// Byte 176: BYTE  Data[164];
// Byte 177: BYTE  Data[165];
// Byte 178: BYTE  Data[166];
// Byte 179: BYTE  Data[167];
// Byte 180: BYTE  Data[168];
// Byte 181: BYTE  Data[169];
// Byte 182: BYTE  Data[170];
// Byte 183: BYTE  Data[171];
// Byte 184: BYTE  Data[172];
// Byte 185: BYTE  Data[173];
// Byte 186: BYTE  Data[174];
// Byte 187: BYTE  Data[175];
// Byte 188: BYTE  Data[176];
// Byte 189: BYTE  Data[177];
// Byte 190: BYTE  Data[178];
// Byte 191: BYTE  Data[179];
// Byte 192: BYTE  Data[180];
// Byte 193: BYTE  Data[181];
// Byte 194: BYTE  Data[182];
// Byte 195: BYTE  Data[183];
// Byte 196: BYTE  Data[184];
// Byte 197: BYTE  Data[185];
// Byte 198: BYTE  Data[186];
// Byte 199: BYTE  Data[187];
// Byte 200: BYTE  Data[188];
// Byte 201: BYTE  Data[189];
VAR
  /// internal index for loops
  _idx : DINT;
END_VAR
// set command parameter 
_command.CmdTyp       :=  CmdType.CallSubprogram;
_command.ExecMode     :=  ExecMode;
_command.ParSeq       := _command.ParSeq;
_command.Priority     :=  Priority;
_command.EmitterID[0] :=  0;
_command.EmitterID[1] :=  0;
_command.EmitterID[2] :=  0;
_command.EmitterID[3] :=  0;
_command.Reserve      :=  0;
_command.ListenerID   := _parCmd.ListenerID;
_command.Reserve      := 0;
_command.JobID        := _parCmd.JobID;
_command.Data         := _parCmd.Data;


// copy command data to header
_cmdHeader := _command;
// call base implementation to copy header to payload buffer
CreateCommandPayload := SUPER^.CreateCommandPayload(AxesGroup := AxesGroup);

// add command.EmitterID[0]
CreateCommandPayload.AddSint(_command.EmitterID[0]);
// add command.EmitterID[1]
CreateCommandPayload.AddSint(_command.EmitterID[1]);
// add command.EmitterID[2]
CreateCommandPayload.AddSint(_command.EmitterID[2]);
// add command.EmitterID[3]
CreateCommandPayload.AddSint(_command.EmitterID[3]);
// add command.ListenerID
CreateCommandPayload.AddSint(_command.ListenerID);
// add command.Reserve
CreateCommandPayload.AddByte(_command.Reserve);
// add command.JobID
CreateCommandPayload.AddUint(_command.JobID);

